// TIA Portal project "deneme1" (V16)

(* hardware
DEVICE "HMI_1"  TP1200 Comfort
   slot 0: "HMI_1"  TP1200 Comfort  6AV2 124-0MC01-0AX0  16.0.0.0
   slot 1: "HMI_RT_1"  TP1200 Comfort  6AV2 124-0MC01-0AX0  16.0.0.0
   slot 5: "HMI_1.IE_CP_1"  PROFINET Interface  16.0.0.0
      slot 1: "PROFINET Interface_1"  PROFINET Interface
         slot 1: "Port_1"  Port
         slot 2: "Port_2"  Port
   slot 7: "HMI_1.MPI/DP_CP_1"  MPI/DP Interface  16.0.0.0
DEVICE "S71500/ET200MP station_1"  S7-1500 station
   slot 0: "Rail_0"  Rack  6ES7 590-1***0-0AA0
   slot 1: "PLC_1"  CPU 1515-2 PN  6ES7 515-2AM00-0AB0  V1.8
      slot 3: "CPU display_1"  6ES7591-1BA00-0AA0
      slot 32768: "PROFINET interface_1"  X1
         slot 32769: "Port_1"  X1 P1
         slot 32770: "Port_2"  X1 P2
      slot 33024: "PROFINET interface_2"  X2
         slot 33025: "Port_1"  X2 P1
*)

// ===== PLC "PLC_1"  CPU 1515-2 PN =====

VAR_GLOBAL   // PLC tag table "Default tag table"
   "BulunduğuKat" AT %MW0 : Int;
   "Asansor0katta" AT %M2.0 : Bool;
   "Asansor1katta" AT %M2.1 : Bool;
   "Asansor3katta" AT %M2.2 : Bool;
   "Asansor2katta" AT %M2.3 : Bool;
   "P_TRIG1" AT %M2.4 : Bool;
   "AsansorAsagı" AT %M2.5 : Bool;
   "P_TRIG2" AT %M2.6 : Bool;
   "AsansorAcKat0" AT %M2.7 : Bool;
   "KapıAcık" AT %M3.0 : Bool;
   "P_TRIG3" AT %M3.1 : Bool;
   "AsansorKapatKat0" AT %M3.2 : Bool;
   "P_TRIG4" AT %M3.3 : Bool;
   "KapıKapalı" AT %M3.4 : Bool;
   "IsıkBariyeri" AT %M3.5 : Bool;
   "0KatDown" AT %M3.6 : Bool;
   "P_TRIG5" AT %M3.7 : Bool;
   "1KatGİT" AT %M4.0 : Bool;
   "2KatGİT" AT %M4.1 : Bool;
   "3KatGİT" AT %M4.2 : Bool;
   "AsansorYukarı" AT %M4.3 : Bool;
   "P_TRIG6" AT %M4.4 : Bool;
   "AsansorAcKat1" AT %M4.5 : Bool;
   "P_TRIG7" AT %M4.6 : Bool;
   "AsansorKapatKat1" AT %M4.7 : Bool;
   "P_TRIG8" AT %M5.0 : Bool;
   "P_TRIG9" AT %M5.1 : Bool;
   "P_TRIG10" AT %M5.2 : Bool;
   "AsansorAcKat2" AT %M5.3 : Bool;
   "P_TRIG11" AT %M5.4 : Bool;
   "P_TRIG12" AT %M5.5 : Bool;
   "AsansorAcKat3" AT %M5.6 : Bool;
   "1Katagit0dan" AT %M5.7 : Bool;
   "2katagit0dan" AT %M6.0 : Bool;
   "3katagit0dan" AT %M6.1 : Bool;
   "P_TRIG13" AT %M6.2 : Bool;
   "P_TRIG14" AT %M6.3 : Bool;
   "P_TRIG15" AT %M6.4 : Bool;
   "P_TRIG16" AT %M6.5 : Bool;
   "P_TRIG17" AT %M6.6 : Bool;
   "AsansorKapatKat2" AT %M6.7 : Bool;
   "AsansorKapatKat3" AT %M7.0 : Bool;
   "P_TRIG18" AT %M7.1 : Bool;
   "P_TRIG19" AT %M7.2 : Bool;
   "P_TRIG20" AT %M7.3 : Bool;
   "P_TRIG21" AT %M7.4 : Bool;
   "1KatDown" AT %M7.5 : Bool;
   "P_TRIG22" AT %M7.6 : Bool;
   "1KatUp" AT %M7.7 : Bool;
   "P_TRIG23" AT %M8.0 : Bool;
   "P_TRIG25" AT %M8.1 : Bool;
   "P_TRIG24" AT %M8.2 : Bool;
   "P_TRIG26" AT %M8.3 : Bool;
   "0KataGit" AT %M8.4 : Bool;
   "2katagit1den" AT %M8.5 : Bool;
   "3katagit1den" AT %M8.6 : Bool;
   "0katagit1den" AT %M8.7 : Bool;
   "P_TRIG27" AT %M9.0 : Bool;
   "P_TRIG28" AT %M9.1 : Bool;
   "P_TRIG29" AT %M9.2 : Bool;
   "P_TRIG30" AT %M9.3 : Bool;
   "P_TRIG31" AT %M9.4 : Bool;
   "P_TRIG32" AT %M9.5 : Bool;
   "P_TRIG33" AT %M9.6 : Bool;
   "P_TRIG34" AT %M9.7 : Bool;
   "P_TRIG35" AT %M10.0 : Bool;
   "P_TRIG36" AT %M10.1 : Bool;
   "P_TRIG37" AT %M10.2 : Bool;
   "P_TRIG38" AT %M10.3 : Bool;
   "P_TRIG39" AT %M10.4 : Bool;
   "P_TRIG40" AT %M10.5 : Bool;
   "Asansorsuan1katta" AT %M10.6 : Bool;
   "Asansorsuan0katta" AT %M10.7 : Bool;
   "P_TRIG41" AT %M11.0 : Bool;
   "P_TRIG42" AT %M11.1 : Bool;
   "P_TRIG43" AT %M11.2 : Bool;
   "P_TRIG44" AT %M11.3 : Bool;
   "P_TRIG45" AT %M11.4 : Bool;
   "P_TRIG46" AT %M11.5 : Bool;
   "P_TRIG47" AT %M11.6 : Bool;
   "P_TRIG48" AT %M11.7 : Bool;
   "P_TRIG49" AT %M12.0 : Bool;
   "P_TRIG50" AT %M12.1 : Bool;
   "P_TRIG51" AT %M12.2 : Bool;
   "P_TRIG52" AT %M12.3 : Bool;
   "P_TRIG53" AT %M12.4 : Bool;
   "P_TRIG54" AT %M12.5 : Bool;
   "P_TRIG55" AT %M12.6 : Bool;
   "P_TRIG56" AT %M12.7 : Bool;
   "deneme1" AT %M13.0 : Bool;
   "P_TRIG100" AT %M13.1 : Bool;
   "P_TRIG101" AT %M13.2 : Bool;
   "P_TRIG102" AT %M13.3 : Bool;
   "kapıacıkset" AT %M13.4 : Bool;
   "P_TRIG103" AT %M13.5 : Bool;
   "P_TRIG104" AT %M13.6 : Bool;
   "P_TRIG107" AT %M13.7 : Bool;
   "P_TRIG108" AT %M14.0 : Bool;
   "P_TRIG106" AT %M14.1 : Bool;
   "P_TRIG105" AT %M14.2 : Bool;
   "P_TRIG111" AT %M14.3 : Bool;
   "P_TRIG110" AT %M14.4 : Bool;
   "P_TRIG109" AT %M14.5 : Bool;
   "P_TRIG114" AT %M14.6 : Bool;
   "P_TRIG113" AT %M14.7 : Bool;
   "P_TRIG112" AT %M15.0 : Bool;
   "P_TRIG120" AT %M15.1 : Bool;
   "P_TRIG115" AT %M15.2 : Bool;
   "P_TRIG116" AT %M15.3 : Bool;
   "P_TRIG117" AT %M15.4 : Bool;
   "P_TRIG118" AT %M15.5 : Bool;
   "P_TRIG119" AT %M15.6 : Bool;
   "P_TRIG126" AT %M15.7 : Bool;
   "P_TRIG121" AT %M16.0 : Bool;
   "P_TRIG122" AT %M16.1 : Bool;
   "P_TRIG123" AT %M16.2 : Bool;
   "P_TRIG124" AT %M16.3 : Bool;
   "P_TRIG125" AT %M16.4 : Bool;
   "P_TRIG127" AT %M16.5 : Bool;
   "P_TRIG128" AT %M16.6 : Bool;
   "P_TRIG129" AT %M16.7 : Bool;
   "Asansorsuan2katta" AT %M17.0 : Bool;
   "P_TRIG130" AT %M17.6 : Bool;
   "P_TRIG131" AT %M17.1 : Bool;
   "P_TRIG132" AT %M17.2 : Bool;
   "P_TRIG133" AT %M17.5 : Bool;
   "P_TRIG134" AT %M17.3 : Bool;
   "P_TRIG135" AT %M17.4 : Bool;
   "3katagit2den" AT %M17.7 : Bool;
   "1katagit2den" AT %M18.0 : Bool;
   "0katagit2den" AT %M18.1 : Bool;
   "P_TRIG138" AT %M18.6 : Bool;
   "P_TRIG136" AT %M18.2 : Bool;
   "P_TRIG137" AT %M18.7 : Bool;
   "P_TRIG139" AT %M19.0 : Bool;
   "P_TRIG140" AT %M18.3 : Bool;
   "P_TRIG141" AT %M18.4 : Bool;
   "P_TRIG142" AT %M18.5 : Bool;
   "P_TRIG144" AT %M19.1 : Bool;
   "P_TRIG143" AT %M19.2 : Bool;
   "P_TRIG145" AT %M19.3 : Bool;
   "P_TRIG146" AT %M19.4 : Bool;
   "P_TRIG147" AT %M19.5 : Bool;
   "P_TRIG148" AT %M19.6 : Bool;
   "P_TRIG149" AT %M20.3 : Bool;
   "P_TRIG150" AT %M19.7 : Bool;
   "P_TRIG151" AT %M20.0 : Bool;
   "P_TRIG152" AT %M20.1 : Bool;
   "P_TRIG153" AT %M20.2 : Bool;
   "P_TRIG154" AT %M20.4 : Bool;
   "P_TRIG155" AT %M20.5 : Bool;
   "P_TRIG156" AT %M20.6 : Bool;
   "3katUp" AT %M20.7 : Bool;
   "Asansorsuan3katta" AT %M21.0 : Bool;
   "2katagit3den" AT %M21.1 : Bool;
   "1katagit3den" AT %M21.2 : Bool;
   "0katagit3den" AT %M21.3 : Bool;
   "P_TRIG164" AT %M21.4 : Bool;
   "P_TRIG163" AT %M22.0 : Bool;
   "P_TRIG162" AT %M21.5 : Bool;
   "P_TRIG161" AT %M21.6 : Bool;
   "P_TRIG160" AT %M21.7 : Bool;
   "P_TRIG171" AT %M22.1 : Bool;
   "P_TRIG170" AT %M22.2 : Bool;
   "P_TRIG169" AT %M22.7 : Bool;
   "P_TRIG168" AT %M22.3 : Bool;
   "P_TRIG167" AT %M22.4 : Bool;
   "P_TRIG166" AT %M22.5 : Bool;
   "P_TRIG165" AT %M22.6 : Bool;
   "P_TRIG172" AT %M23.0 : Bool;
   "P_TRIG173" AT %M23.1 : Bool;
   "P_TRIG174" AT %M23.2 : Bool;
   "P_TRIG175" AT %M23.3 : Bool;
   "P_TRIG176" AT %M23.4 : Bool;
   "P_TRIG177" AT %M23.5 : Bool;
   "P_TRIG178" AT %M23.6 : Bool;
   "P_TRIG179" AT %M23.7 : Bool;
   "P_TRIG180" AT %M24.0 : Bool;
   "P_TRIG181" AT %M24.1 : Bool;
   "P_TRIG182" AT %M24.2 : Bool;
   "P_TRIG183" AT %M24.3 : Bool;
   "P_TRIG184" AT %M24.4 : Bool;
   "P_TRIG185" AT %M24.5 : Bool;
   "P_TRIG186" AT %M24.6 : Bool;
   "2KatDown" AT %M24.7 : Bool;
   "2KatUp" AT %M25.0 : Bool;
END_VAR

ORGANIZATION_BLOCK "Main"   // OB1, LAD, ProgramCycle
TITLE = "Main Program Sweep (Cycle)"
{ S7_Optimized_Access := 'TRUE' }
VERSION : 0.1
   VAR_INPUT
      Initial_Call : Bool;   // Initial call of this OB
      Remanence : Bool;   // =True, if remanent data are available
   END_VAR
   VAR_TEMP   // added for the SCL form of the ladder/FBD networks
      _w1 : Bool;
      _w2 : Bool;
      _w3 : Bool;
      _w4 : Bool;
      _w5 : Bool;
      _w6 : Bool;
      _w7 : Bool;
      _w8 : Bool;
      _w9 : Bool;
      _w10 : Bool;
      _w11 : Bool;
      _w12 : Bool;
      _w13 : Bool;
      _w14 : Bool;
      _w15 : Bool;
      _w16 : Bool;
      _w17 : Bool;
      _w18 : Bool;
      _w19 : Bool;
      _w20 : Bool;
      _w21 : Bool;
      _w22 : Bool;
      _w23 : Bool;
      _w24 : Bool;
      _w25 : Bool;
      _w26 : Bool;
      _w27 : Bool;
      _w28 : Bool;
      _w29 : Bool;
      _w30 : Bool;
      _w31 : Bool;
      _w32 : Bool;
      _w33 : Bool;
      _w34 : Bool;
      _w35 : Bool;
      _w36 : Bool;
      _w37 : Bool;
      _w38 : Bool;
      _w39 : Bool;
      _w40 : Bool;
      _w41 : Bool;
      _w42 : Bool;
      _w43 : Bool;
      _w44 : Bool;
      _w45 : Bool;
      _w46 : Bool;
      _w47 : Bool;
      _w48 : Bool;
      _w49 : Bool;
      _w50 : Bool;
      _w51 : Bool;
      _w52 : Bool;
      _w53 : Bool;
      _w54 : Bool;
      _w55 : Bool;
   END_VAR
BEGIN

REGION Network 1: 0 a bas 1 2 3 den asansör gelsin
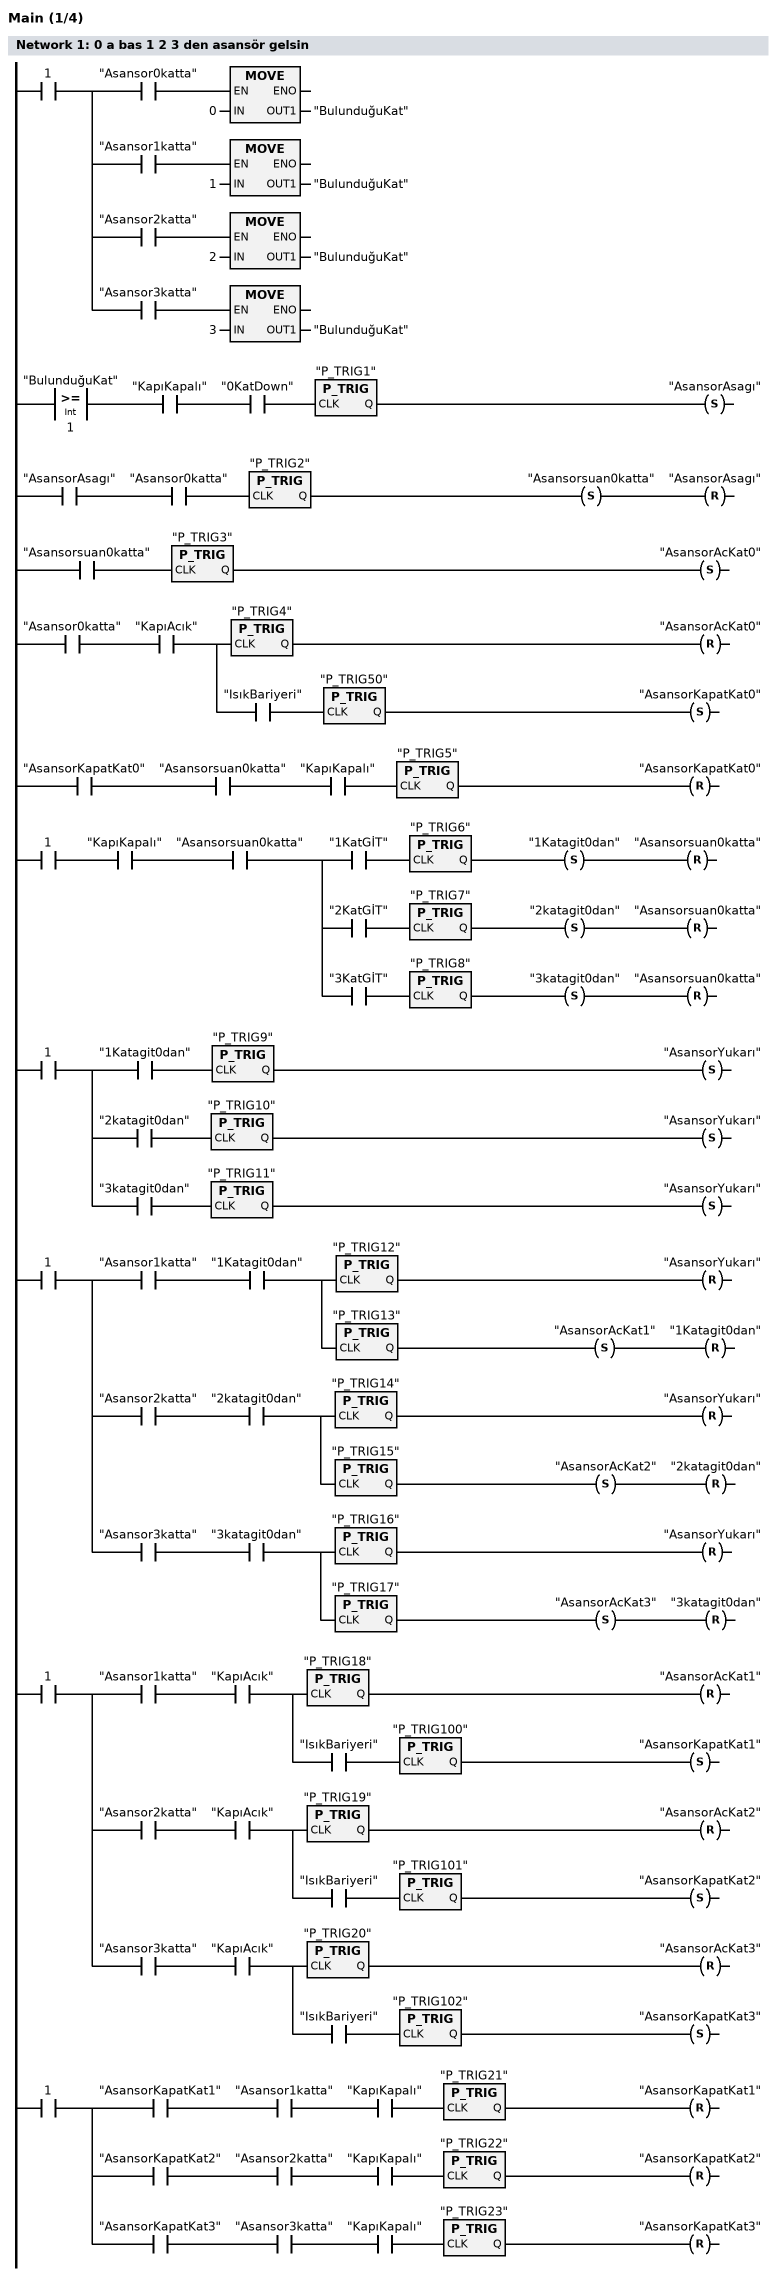
   RUNG wire#powerrail
      Contact( 1 )
      wire#w1
      Contact( "Asansor0katta" )
      Move(in := 0, out1 => "BulunduğuKat")
   END_RUNG
   RUNG wire#w1
      Contact( "Asansor1katta" )
      Move(in := 1, out1 => "BulunduğuKat")
   END_RUNG
   RUNG wire#w1
      Contact( "Asansor2katta" )
      Move(in := 2, out1 => "BulunduğuKat")
   END_RUNG
   RUNG wire#w1
      Contact( "Asansor3katta" )
      Move(in := 3, out1 => "BulunduğuKat")
   END_RUNG
   RUNG wire#powerrail
      { S7_Templates := "SrcType := Int" } GE_Contact(in1 := "BulunduğuKat", in2 := 1)
      Contact( "KapıKapalı" )
      Contact( "0KatDown" )
      P_Trig( "P_TRIG1" )
      S_Coil( "AsansorAsagı" )
   END_RUNG
   RUNG wire#powerrail
      Contact( "AsansorAsagı" )
      Contact( "Asansor0katta" )
      P_Trig( "P_TRIG2" )
      S_Coil( "Asansorsuan0katta" )
      R_Coil( "AsansorAsagı" )
   END_RUNG
   RUNG wire#powerrail
      Contact( "Asansorsuan0katta" )
      P_Trig( "P_TRIG3" )
      S_Coil( "AsansorAcKat0" )
   END_RUNG
   RUNG wire#powerrail
      Contact( "Asansor0katta" )
      Contact( "KapıAcık" )
      wire#w2
      P_Trig( "P_TRIG4" )
      R_Coil( "AsansorAcKat0" )
   END_RUNG
   RUNG wire#w2
      Contact( "IsıkBariyeri" )
      P_Trig( "P_TRIG50" )
      S_Coil( "AsansorKapatKat0" )
   END_RUNG
   RUNG wire#powerrail
      Contact( "AsansorKapatKat0" )
      Contact( "Asansorsuan0katta" )
      Contact( "KapıKapalı" )
      P_Trig( "P_TRIG5" )
      R_Coil( "AsansorKapatKat0" )
   END_RUNG
   RUNG wire#powerrail
      Contact( 1 )
      Contact( "KapıKapalı" )
      Contact( "Asansorsuan0katta" )
      wire#w3
      Contact( "1KatGİT" )
      P_Trig( "P_TRIG6" )
      S_Coil( "1Katagit0dan" )
      R_Coil( "Asansorsuan0katta" )
   END_RUNG
   RUNG wire#w3
      Contact( "2KatGİT" )
      P_Trig( "P_TRIG7" )
      S_Coil( "2katagit0dan" )
      R_Coil( "Asansorsuan0katta" )
   END_RUNG
   RUNG wire#w3
      Contact( "3KatGİT" )
      P_Trig( "P_TRIG8" )
      S_Coil( "3katagit0dan" )
      R_Coil( "Asansorsuan0katta" )
   END_RUNG
   RUNG wire#powerrail
      Contact( 1 )
      wire#w4
      Contact( "1Katagit0dan" )
      P_Trig( "P_TRIG9" )
      S_Coil( "AsansorYukarı" )
   END_RUNG
   RUNG wire#w4
      Contact( "2katagit0dan" )
      P_Trig( "P_TRIG10" )
      S_Coil( "AsansorYukarı" )
   END_RUNG
   RUNG wire#w4
      Contact( "3katagit0dan" )
      P_Trig( "P_TRIG11" )
      S_Coil( "AsansorYukarı" )
   END_RUNG
   RUNG wire#powerrail
      Contact( 1 )
      wire#w5
      Contact( "Asansor1katta" )
      Contact( "1Katagit0dan" )
      wire#w6
      P_Trig( "P_TRIG12" )
      R_Coil( "AsansorYukarı" )
   END_RUNG
   RUNG wire#w6
      P_Trig( "P_TRIG13" )
      S_Coil( "AsansorAcKat1" )
      R_Coil( "1Katagit0dan" )
   END_RUNG
   RUNG wire#w5
      Contact( "Asansor2katta" )
      Contact( "2katagit0dan" )
      wire#w7
      P_Trig( "P_TRIG14" )
      R_Coil( "AsansorYukarı" )
   END_RUNG
   RUNG wire#w7
      P_Trig( "P_TRIG15" )
      S_Coil( "AsansorAcKat2" )
      R_Coil( "2katagit0dan" )
   END_RUNG
   RUNG wire#w5
      Contact( "Asansor3katta" )
      Contact( "3katagit0dan" )
      wire#w8
      P_Trig( "P_TRIG16" )
      R_Coil( "AsansorYukarı" )
   END_RUNG
   RUNG wire#w8
      P_Trig( "P_TRIG17" )
      S_Coil( "AsansorAcKat3" )
      R_Coil( "3katagit0dan" )
   END_RUNG
   RUNG wire#powerrail
      Contact( 1 )
      wire#w9
      Contact( "Asansor1katta" )
      Contact( "KapıAcık" )
      wire#w10
      P_Trig( "P_TRIG18" )
      R_Coil( "AsansorAcKat1" )
   END_RUNG
   RUNG wire#w10
      Contact( "IsıkBariyeri" )
      P_Trig( "P_TRIG100" )
      S_Coil( "AsansorKapatKat1" )
   END_RUNG
   RUNG wire#w9
      Contact( "Asansor2katta" )
      Contact( "KapıAcık" )
      wire#w11
      P_Trig( "P_TRIG19" )
      R_Coil( "AsansorAcKat2" )
   END_RUNG
   RUNG wire#w11
      Contact( "IsıkBariyeri" )
      P_Trig( "P_TRIG101" )
      S_Coil( "AsansorKapatKat2" )
   END_RUNG
   RUNG wire#w9
      Contact( "Asansor3katta" )
      Contact( "KapıAcık" )
      wire#w12
      P_Trig( "P_TRIG20" )
      R_Coil( "AsansorAcKat3" )
   END_RUNG
   RUNG wire#w12
      Contact( "IsıkBariyeri" )
      P_Trig( "P_TRIG102" )
      S_Coil( "AsansorKapatKat3" )
   END_RUNG
   RUNG wire#powerrail
      Contact( 1 )
      wire#w13
      Contact( "AsansorKapatKat1" )
      Contact( "Asansor1katta" )
      Contact( "KapıKapalı" )
      P_Trig( "P_TRIG21" )
      R_Coil( "AsansorKapatKat1" )
   END_RUNG
   RUNG wire#w13
      Contact( "AsansorKapatKat2" )
      Contact( "Asansor2katta" )
      Contact( "KapıKapalı" )
      P_Trig( "P_TRIG22" )
      R_Coil( "AsansorKapatKat2" )
   END_RUNG
   RUNG wire#w13
      Contact( "AsansorKapatKat3" )
      Contact( "Asansor3katta" )
      Contact( "KapıKapalı" )
      P_Trig( "P_TRIG23" )
      R_Coil( "AsansorKapatKat3" )
   END_RUNG
   // the same network as SCL:
   IF 1 AND "Asansor0katta" THEN "BulunduğuKat" := 0; END_IF;
   IF 1 AND "Asansor1katta" THEN "BulunduğuKat" := 1; END_IF;
   IF 1 AND "Asansor2katta" THEN "BulunduğuKat" := 2; END_IF;
   IF 1 AND "Asansor3katta" THEN "BulunduğuKat" := 3; END_IF;
   #_w1 := ("BulunduğuKat" >= 1) AND "KapıKapalı" AND "0KatDown";
   #_w2 := #_w1 AND NOT "P_TRIG1";   // rising edge
   "P_TRIG1" := #_w1;
   IF #_w2 THEN "AsansorAsagı" := TRUE; END_IF;
   #_w3 := "AsansorAsagı" AND "Asansor0katta";
   #_w4 := #_w3 AND NOT "P_TRIG2";   // rising edge
   "P_TRIG2" := #_w3;
   IF #_w4 THEN
       "Asansorsuan0katta" := TRUE;
       "AsansorAsagı" := FALSE;
   END_IF;
   #_w5 := "Asansorsuan0katta" AND NOT "P_TRIG3";   // rising edge
   "P_TRIG3" := "Asansorsuan0katta";
   IF #_w5 THEN "AsansorAcKat0" := TRUE; END_IF;
   #_w6 := "Asansor0katta" AND "KapıAcık";
   #_w7 := #_w6 AND NOT "P_TRIG4";   // rising edge
   "P_TRIG4" := #_w6;
   IF #_w7 THEN "AsansorAcKat0" := FALSE; END_IF;
   #_w8 := #_w6 AND "IsıkBariyeri";
   #_w9 := #_w8 AND NOT "P_TRIG50";   // rising edge
   "P_TRIG50" := #_w8;
   IF #_w9 THEN "AsansorKapatKat0" := TRUE; END_IF;
   #_w10 := "AsansorKapatKat0" AND "Asansorsuan0katta" AND "KapıKapalı";
   #_w11 := #_w10 AND NOT "P_TRIG5";   // rising edge
   "P_TRIG5" := #_w10;
   IF #_w11 THEN "AsansorKapatKat0" := FALSE; END_IF;
   #_w12 := 1 AND "KapıKapalı" AND "Asansorsuan0katta";
   #_w13 := #_w12 AND "1KatGİT";
   #_w14 := #_w13 AND NOT "P_TRIG6";   // rising edge
   "P_TRIG6" := #_w13;
   IF #_w14 THEN
       "1Katagit0dan" := TRUE;
       "Asansorsuan0katta" := FALSE;
   END_IF;
   #_w15 := #_w12 AND "2KatGİT";
   #_w16 := #_w15 AND NOT "P_TRIG7";   // rising edge
   "P_TRIG7" := #_w15;
   IF #_w16 THEN
       "2katagit0dan" := TRUE;
       "Asansorsuan0katta" := FALSE;
   END_IF;
   #_w17 := #_w12 AND "3KatGİT";
   #_w18 := #_w17 AND NOT "P_TRIG8";   // rising edge
   "P_TRIG8" := #_w17;
   IF #_w18 THEN
       "3katagit0dan" := TRUE;
       "Asansorsuan0katta" := FALSE;
   END_IF;
   #_w19 := 1 AND "1Katagit0dan";
   #_w20 := #_w19 AND NOT "P_TRIG9";   // rising edge
   "P_TRIG9" := #_w19;
   IF #_w20 THEN "AsansorYukarı" := TRUE; END_IF;
   #_w21 := 1 AND "2katagit0dan";
   #_w22 := #_w21 AND NOT "P_TRIG10";   // rising edge
   "P_TRIG10" := #_w21;
   IF #_w22 THEN "AsansorYukarı" := TRUE; END_IF;
   #_w23 := 1 AND "3katagit0dan";
   #_w24 := #_w23 AND NOT "P_TRIG11";   // rising edge
   "P_TRIG11" := #_w23;
   IF #_w24 THEN "AsansorYukarı" := TRUE; END_IF;
   #_w25 := 1 AND "Asansor1katta" AND "1Katagit0dan";
   #_w26 := #_w25 AND NOT "P_TRIG12";   // rising edge
   "P_TRIG12" := #_w25;
   IF #_w26 THEN "AsansorYukarı" := FALSE; END_IF;
   #_w27 := #_w25 AND NOT "P_TRIG13";   // rising edge
   "P_TRIG13" := #_w25;
   IF #_w27 THEN
       "AsansorAcKat1" := TRUE;
       "1Katagit0dan" := FALSE;
   END_IF;
   #_w28 := 1 AND "Asansor2katta" AND "2katagit0dan";
   #_w29 := #_w28 AND NOT "P_TRIG14";   // rising edge
   "P_TRIG14" := #_w28;
   IF #_w29 THEN "AsansorYukarı" := FALSE; END_IF;
   #_w30 := #_w28 AND NOT "P_TRIG15";   // rising edge
   "P_TRIG15" := #_w28;
   IF #_w30 THEN
       "AsansorAcKat2" := TRUE;
       "2katagit0dan" := FALSE;
   END_IF;
   #_w31 := 1 AND "Asansor3katta" AND "3katagit0dan";
   #_w32 := #_w31 AND NOT "P_TRIG16";   // rising edge
   "P_TRIG16" := #_w31;
   IF #_w32 THEN "AsansorYukarı" := FALSE; END_IF;
   #_w33 := #_w31 AND NOT "P_TRIG17";   // rising edge
   "P_TRIG17" := #_w31;
   IF #_w33 THEN
       "AsansorAcKat3" := TRUE;
       "3katagit0dan" := FALSE;
   END_IF;
   #_w34 := 1 AND "Asansor1katta" AND "KapıAcık";
   #_w35 := #_w34 AND NOT "P_TRIG18";   // rising edge
   "P_TRIG18" := #_w34;
   IF #_w35 THEN "AsansorAcKat1" := FALSE; END_IF;
   #_w36 := #_w34 AND "IsıkBariyeri";
   #_w37 := #_w36 AND NOT "P_TRIG100";   // rising edge
   "P_TRIG100" := #_w36;
   IF #_w37 THEN "AsansorKapatKat1" := TRUE; END_IF;
   #_w38 := 1 AND "Asansor2katta" AND "KapıAcık";
   #_w39 := #_w38 AND NOT "P_TRIG19";   // rising edge
   "P_TRIG19" := #_w38;
   IF #_w39 THEN "AsansorAcKat2" := FALSE; END_IF;
   #_w40 := #_w38 AND "IsıkBariyeri";
   #_w41 := #_w40 AND NOT "P_TRIG101";   // rising edge
   "P_TRIG101" := #_w40;
   IF #_w41 THEN "AsansorKapatKat2" := TRUE; END_IF;
   #_w42 := 1 AND "Asansor3katta" AND "KapıAcık";
   #_w43 := #_w42 AND NOT "P_TRIG20";   // rising edge
   "P_TRIG20" := #_w42;
   IF #_w43 THEN "AsansorAcKat3" := FALSE; END_IF;
   #_w44 := #_w42 AND "IsıkBariyeri";
   #_w45 := #_w44 AND NOT "P_TRIG102";   // rising edge
   "P_TRIG102" := #_w44;
   IF #_w45 THEN "AsansorKapatKat3" := TRUE; END_IF;
   #_w46 := 1 AND "AsansorKapatKat1" AND "Asansor1katta" AND "KapıKapalı";
   #_w47 := #_w46 AND NOT "P_TRIG21";   // rising edge
   "P_TRIG21" := #_w46;
   IF #_w47 THEN "AsansorKapatKat1" := FALSE; END_IF;
   #_w48 := 1 AND "AsansorKapatKat2" AND "Asansor2katta" AND "KapıKapalı";
   #_w49 := #_w48 AND NOT "P_TRIG22";   // rising edge
   "P_TRIG22" := #_w48;
   IF #_w49 THEN "AsansorKapatKat2" := FALSE; END_IF;
   #_w50 := 1 AND "AsansorKapatKat3" AND "Asansor3katta" AND "KapıKapalı";
   #_w51 := #_w50 AND NOT "P_TRIG23";   // rising edge
   "P_TRIG23" := #_w50;
   IF #_w51 THEN "AsansorKapatKat3" := FALSE; END_IF;
END_REGION

REGION Network 2: 1 katda iken 0 dan çağırma veya 1 katda iken 2 ve 3 den cağırma
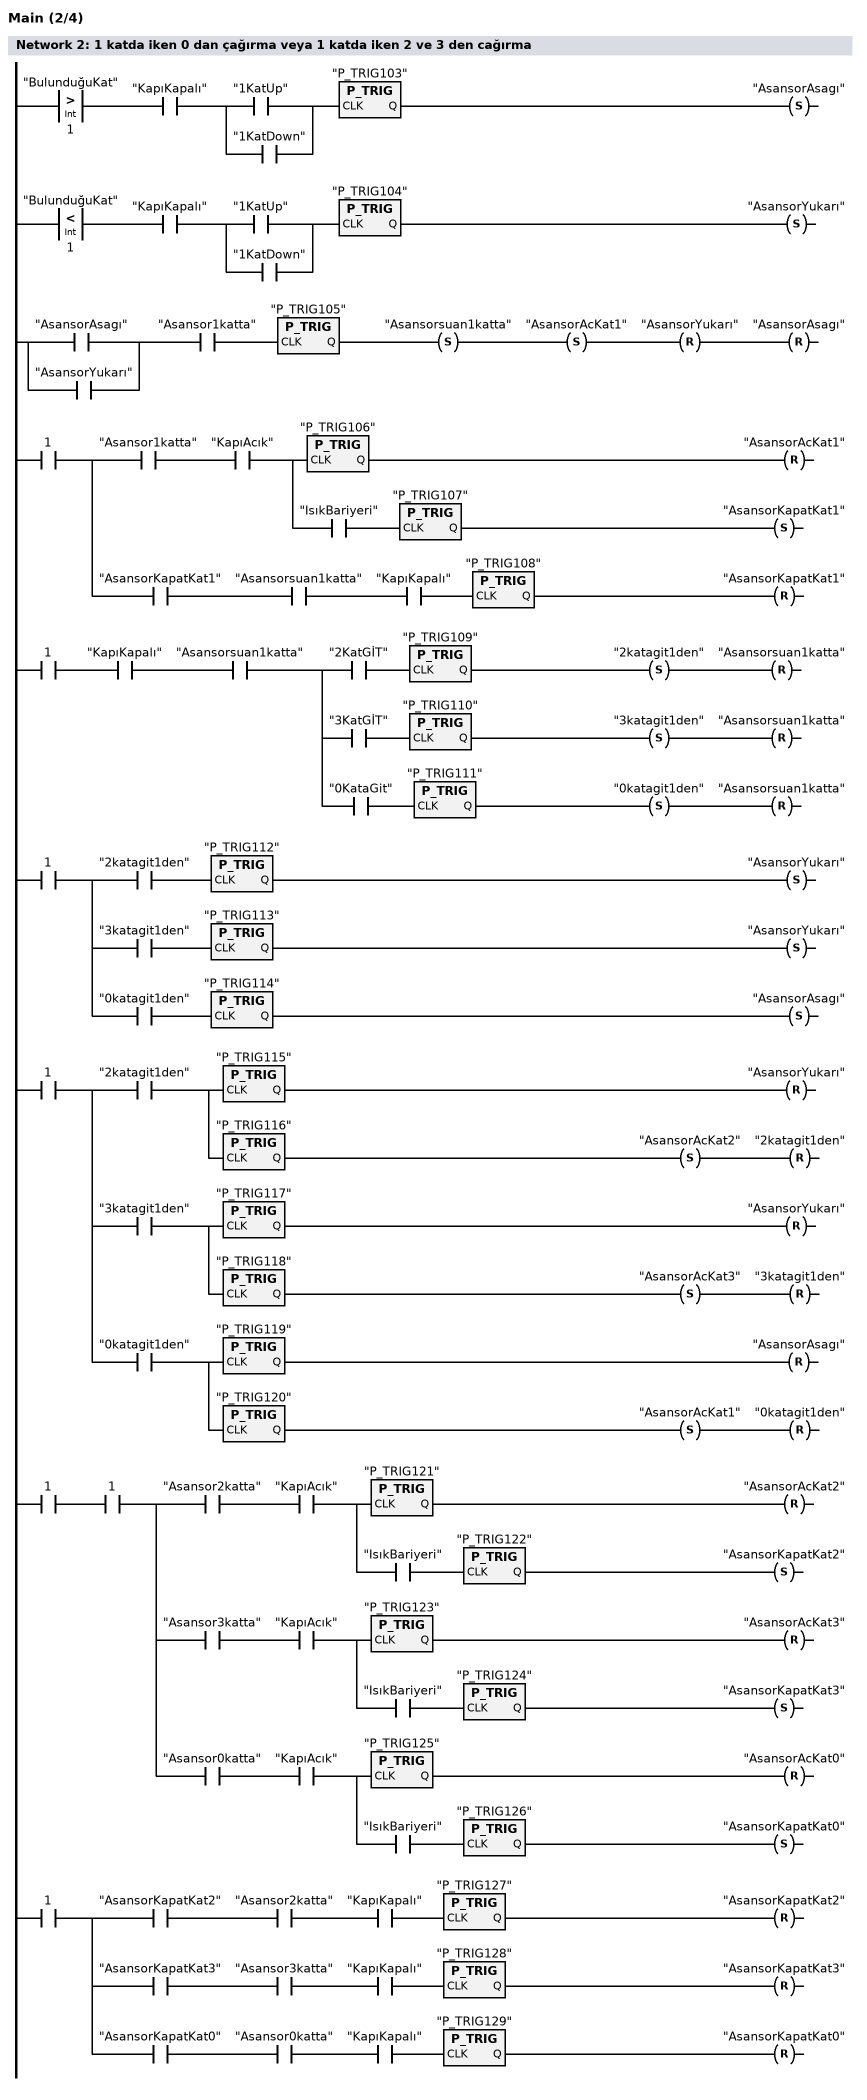
   RUNG wire#powerrail
      { S7_Templates := "SrcType := Int" } GT_Contact(in1 := "BulunduğuKat", in2 := 1)
      Contact( "KapıKapalı" )
      wire#w1
      Contact( "1KatUp" )
      wire#w2
      P_Trig( "P_TRIG103" )
      S_Coil( "AsansorAsagı" )
   END_RUNG
   RUNG wire#w1
      Contact( "1KatDown" )
   END_RUNG wire#w2
   RUNG wire#powerrail
      { S7_Templates := "SrcType := Int" } LT_Contact(in1 := "BulunduğuKat", in2 := 1)
      Contact( "KapıKapalı" )
      wire#w3
      Contact( "1KatUp" )
      wire#w4
      P_Trig( "P_TRIG104" )
      S_Coil( "AsansorYukarı" )
   END_RUNG
   RUNG wire#w3
      Contact( "1KatDown" )
   END_RUNG wire#w4
   RUNG wire#powerrail
      Contact( "AsansorAsagı" )
      wire#w5
      Contact( "Asansor1katta" )
      P_Trig( "P_TRIG105" )
      S_Coil( "Asansorsuan1katta" )
      S_Coil( "AsansorAcKat1" )
      R_Coil( "AsansorYukarı" )
      R_Coil( "AsansorAsagı" )
   END_RUNG
   RUNG wire#powerrail
      Contact( "AsansorYukarı" )
   END_RUNG wire#w5
   RUNG wire#powerrail
      Contact( 1 )
      wire#w6
      Contact( "Asansor1katta" )
      Contact( "KapıAcık" )
      wire#w7
      P_Trig( "P_TRIG106" )
      R_Coil( "AsansorAcKat1" )
   END_RUNG
   RUNG wire#w7
      Contact( "IsıkBariyeri" )
      P_Trig( "P_TRIG107" )
      S_Coil( "AsansorKapatKat1" )
   END_RUNG
   RUNG wire#w6
      Contact( "AsansorKapatKat1" )
      Contact( "Asansorsuan1katta" )
      Contact( "KapıKapalı" )
      P_Trig( "P_TRIG108" )
      R_Coil( "AsansorKapatKat1" )
   END_RUNG
   RUNG wire#powerrail
      Contact( 1 )
      Contact( "KapıKapalı" )
      Contact( "Asansorsuan1katta" )
      wire#w8
      Contact( "2KatGİT" )
      P_Trig( "P_TRIG109" )
      S_Coil( "2katagit1den" )
      R_Coil( "Asansorsuan1katta" )
   END_RUNG
   RUNG wire#w8
      Contact( "3KatGİT" )
      P_Trig( "P_TRIG110" )
      S_Coil( "3katagit1den" )
      R_Coil( "Asansorsuan1katta" )
   END_RUNG
   RUNG wire#w8
      Contact( "0KataGit" )
      P_Trig( "P_TRIG111" )
      S_Coil( "0katagit1den" )
      R_Coil( "Asansorsuan1katta" )
   END_RUNG
   RUNG wire#powerrail
      Contact( 1 )
      wire#w9
      Contact( "2katagit1den" )
      P_Trig( "P_TRIG112" )
      S_Coil( "AsansorYukarı" )
   END_RUNG
   RUNG wire#w9
      Contact( "3katagit1den" )
      P_Trig( "P_TRIG113" )
      S_Coil( "AsansorYukarı" )
   END_RUNG
   RUNG wire#w9
      Contact( "0katagit1den" )
      P_Trig( "P_TRIG114" )
      S_Coil( "AsansorAsagı" )
   END_RUNG
   RUNG wire#powerrail
      Contact( 1 )
      wire#w10
      Contact( "2katagit1den" )
      wire#w11
      P_Trig( "P_TRIG115" )
      R_Coil( "AsansorYukarı" )
   END_RUNG
   RUNG wire#w11
      P_Trig( "P_TRIG116" )
      S_Coil( "AsansorAcKat2" )
      R_Coil( "2katagit1den" )
   END_RUNG
   RUNG wire#w10
      Contact( "3katagit1den" )
      wire#w12
      P_Trig( "P_TRIG117" )
      R_Coil( "AsansorYukarı" )
   END_RUNG
   RUNG wire#w12
      P_Trig( "P_TRIG118" )
      S_Coil( "AsansorAcKat3" )
      R_Coil( "3katagit1den" )
   END_RUNG
   RUNG wire#w10
      Contact( "0katagit1den" )
      wire#w13
      P_Trig( "P_TRIG119" )
      R_Coil( "AsansorAsagı" )
   END_RUNG
   RUNG wire#w13
      P_Trig( "P_TRIG120" )
      S_Coil( "AsansorAcKat1" )
      R_Coil( "0katagit1den" )
   END_RUNG
   RUNG wire#powerrail
      Contact( 1 )
      Contact( 1 )
      wire#w14
      Contact( "Asansor2katta" )
      Contact( "KapıAcık" )
      wire#w15
      P_Trig( "P_TRIG121" )
      R_Coil( "AsansorAcKat2" )
   END_RUNG
   RUNG wire#w15
      Contact( "IsıkBariyeri" )
      P_Trig( "P_TRIG122" )
      S_Coil( "AsansorKapatKat2" )
   END_RUNG
   RUNG wire#w14
      Contact( "Asansor3katta" )
      Contact( "KapıAcık" )
      wire#w16
      P_Trig( "P_TRIG123" )
      R_Coil( "AsansorAcKat3" )
   END_RUNG
   RUNG wire#w16
      Contact( "IsıkBariyeri" )
      P_Trig( "P_TRIG124" )
      S_Coil( "AsansorKapatKat3" )
   END_RUNG
   RUNG wire#w14
      Contact( "Asansor0katta" )
      Contact( "KapıAcık" )
      wire#w17
      P_Trig( "P_TRIG125" )
      R_Coil( "AsansorAcKat0" )
   END_RUNG
   RUNG wire#w17
      Contact( "IsıkBariyeri" )
      P_Trig( "P_TRIG126" )
      S_Coil( "AsansorKapatKat0" )
   END_RUNG
   RUNG wire#powerrail
      Contact( 1 )
      wire#w18
      Contact( "AsansorKapatKat2" )
      Contact( "Asansor2katta" )
      Contact( "KapıKapalı" )
      P_Trig( "P_TRIG127" )
      R_Coil( "AsansorKapatKat2" )
   END_RUNG
   RUNG wire#w18
      Contact( "AsansorKapatKat3" )
      Contact( "Asansor3katta" )
      Contact( "KapıKapalı" )
      P_Trig( "P_TRIG128" )
      R_Coil( "AsansorKapatKat3" )
   END_RUNG
   RUNG wire#w18
      Contact( "AsansorKapatKat0" )
      Contact( "Asansor0katta" )
      Contact( "KapıKapalı" )
      P_Trig( "P_TRIG129" )
      R_Coil( "AsansorKapatKat0" )
   END_RUNG
   // the same network as SCL:
   #_w1 := ("BulunduğuKat" > 1) AND "KapıKapalı" AND ("1KatUp" OR "1KatDown");
   #_w2 := #_w1 AND NOT "P_TRIG103";   // rising edge
   "P_TRIG103" := #_w1;
   IF #_w2 THEN "AsansorAsagı" := TRUE; END_IF;
   #_w3 := ("BulunduğuKat" < 1) AND "KapıKapalı" AND ("1KatUp" OR "1KatDown");
   #_w4 := #_w3 AND NOT "P_TRIG104";   // rising edge
   "P_TRIG104" := #_w3;
   IF #_w4 THEN "AsansorYukarı" := TRUE; END_IF;
   #_w5 := ("AsansorAsagı" OR "AsansorYukarı") AND "Asansor1katta";
   #_w6 := #_w5 AND NOT "P_TRIG105";   // rising edge
   "P_TRIG105" := #_w5;
   IF #_w6 THEN
       "Asansorsuan1katta" := TRUE;
       "AsansorAcKat1" := TRUE;
       "AsansorYukarı" := FALSE;
       "AsansorAsagı" := FALSE;
   END_IF;
   #_w7 := 1 AND "Asansor1katta" AND "KapıAcık";
   #_w8 := #_w7 AND NOT "P_TRIG106";   // rising edge
   "P_TRIG106" := #_w7;
   IF #_w8 THEN "AsansorAcKat1" := FALSE; END_IF;
   #_w9 := #_w7 AND "IsıkBariyeri";
   #_w10 := #_w9 AND NOT "P_TRIG107";   // rising edge
   "P_TRIG107" := #_w9;
   IF #_w10 THEN "AsansorKapatKat1" := TRUE; END_IF;
   #_w11 := 1 AND "AsansorKapatKat1" AND "Asansorsuan1katta" AND "KapıKapalı";
   #_w12 := #_w11 AND NOT "P_TRIG108";   // rising edge
   "P_TRIG108" := #_w11;
   IF #_w12 THEN "AsansorKapatKat1" := FALSE; END_IF;
   #_w13 := 1 AND "KapıKapalı" AND "Asansorsuan1katta";
   #_w14 := #_w13 AND "2KatGİT";
   #_w15 := #_w14 AND NOT "P_TRIG109";   // rising edge
   "P_TRIG109" := #_w14;
   IF #_w15 THEN
       "2katagit1den" := TRUE;
       "Asansorsuan1katta" := FALSE;
   END_IF;
   #_w16 := #_w13 AND "3KatGİT";
   #_w17 := #_w16 AND NOT "P_TRIG110";   // rising edge
   "P_TRIG110" := #_w16;
   IF #_w17 THEN
       "3katagit1den" := TRUE;
       "Asansorsuan1katta" := FALSE;
   END_IF;
   #_w18 := #_w13 AND "0KataGit";
   #_w19 := #_w18 AND NOT "P_TRIG111";   // rising edge
   "P_TRIG111" := #_w18;
   IF #_w19 THEN
       "0katagit1den" := TRUE;
       "Asansorsuan1katta" := FALSE;
   END_IF;
   #_w20 := 1 AND "2katagit1den";
   #_w21 := #_w20 AND NOT "P_TRIG112";   // rising edge
   "P_TRIG112" := #_w20;
   IF #_w21 THEN "AsansorYukarı" := TRUE; END_IF;
   #_w22 := 1 AND "3katagit1den";
   #_w23 := #_w22 AND NOT "P_TRIG113";   // rising edge
   "P_TRIG113" := #_w22;
   IF #_w23 THEN "AsansorYukarı" := TRUE; END_IF;
   #_w24 := 1 AND "0katagit1den";
   #_w25 := #_w24 AND NOT "P_TRIG114";   // rising edge
   "P_TRIG114" := #_w24;
   IF #_w25 THEN "AsansorAsagı" := TRUE; END_IF;
   #_w26 := 1 AND "2katagit1den";
   #_w27 := #_w26 AND NOT "P_TRIG115";   // rising edge
   "P_TRIG115" := #_w26;
   IF #_w27 THEN "AsansorYukarı" := FALSE; END_IF;
   #_w28 := #_w26 AND NOT "P_TRIG116";   // rising edge
   "P_TRIG116" := #_w26;
   IF #_w28 THEN
       "AsansorAcKat2" := TRUE;
       "2katagit1den" := FALSE;
   END_IF;
   #_w29 := 1 AND "3katagit1den";
   #_w30 := #_w29 AND NOT "P_TRIG117";   // rising edge
   "P_TRIG117" := #_w29;
   IF #_w30 THEN "AsansorYukarı" := FALSE; END_IF;
   #_w31 := #_w29 AND NOT "P_TRIG118";   // rising edge
   "P_TRIG118" := #_w29;
   IF #_w31 THEN
       "AsansorAcKat3" := TRUE;
       "3katagit1den" := FALSE;
   END_IF;
   #_w32 := 1 AND "0katagit1den";
   #_w33 := #_w32 AND NOT "P_TRIG119";   // rising edge
   "P_TRIG119" := #_w32;
   IF #_w33 THEN "AsansorAsagı" := FALSE; END_IF;
   #_w34 := #_w32 AND NOT "P_TRIG120";   // rising edge
   "P_TRIG120" := #_w32;
   IF #_w34 THEN
       "AsansorAcKat1" := TRUE;
       "0katagit1den" := FALSE;
   END_IF;
   #_w35 := 1 AND 1;
   #_w36 := #_w35 AND "Asansor2katta" AND "KapıAcık";
   #_w37 := #_w36 AND NOT "P_TRIG121";   // rising edge
   "P_TRIG121" := #_w36;
   IF #_w37 THEN "AsansorAcKat2" := FALSE; END_IF;
   #_w38 := #_w36 AND "IsıkBariyeri";
   #_w39 := #_w38 AND NOT "P_TRIG122";   // rising edge
   "P_TRIG122" := #_w38;
   IF #_w39 THEN "AsansorKapatKat2" := TRUE; END_IF;
   #_w40 := #_w35 AND "Asansor3katta" AND "KapıAcık";
   #_w41 := #_w40 AND NOT "P_TRIG123";   // rising edge
   "P_TRIG123" := #_w40;
   IF #_w41 THEN "AsansorAcKat3" := FALSE; END_IF;
   #_w42 := #_w40 AND "IsıkBariyeri";
   #_w43 := #_w42 AND NOT "P_TRIG124";   // rising edge
   "P_TRIG124" := #_w42;
   IF #_w43 THEN "AsansorKapatKat3" := TRUE; END_IF;
   #_w44 := #_w35 AND "Asansor0katta" AND "KapıAcık";
   #_w45 := #_w44 AND NOT "P_TRIG125";   // rising edge
   "P_TRIG125" := #_w44;
   IF #_w45 THEN "AsansorAcKat0" := FALSE; END_IF;
   #_w46 := #_w44 AND "IsıkBariyeri";
   #_w47 := #_w46 AND NOT "P_TRIG126";   // rising edge
   "P_TRIG126" := #_w46;
   IF #_w47 THEN "AsansorKapatKat0" := TRUE; END_IF;
   #_w48 := 1 AND "AsansorKapatKat2" AND "Asansor2katta" AND "KapıKapalı";
   #_w49 := #_w48 AND NOT "P_TRIG127";   // rising edge
   "P_TRIG127" := #_w48;
   IF #_w49 THEN "AsansorKapatKat2" := FALSE; END_IF;
   #_w50 := 1 AND "AsansorKapatKat3" AND "Asansor3katta" AND "KapıKapalı";
   #_w51 := #_w50 AND NOT "P_TRIG128";   // rising edge
   "P_TRIG128" := #_w50;
   IF #_w51 THEN "AsansorKapatKat3" := FALSE; END_IF;
   #_w52 := 1 AND "AsansorKapatKat0" AND "Asansor0katta" AND "KapıKapalı";
   #_w53 := #_w52 AND NOT "P_TRIG129";   // rising edge
   "P_TRIG129" := #_w52;
   IF #_w53 THEN "AsansorKapatKat0" := FALSE; END_IF;
END_REGION

REGION Network 3
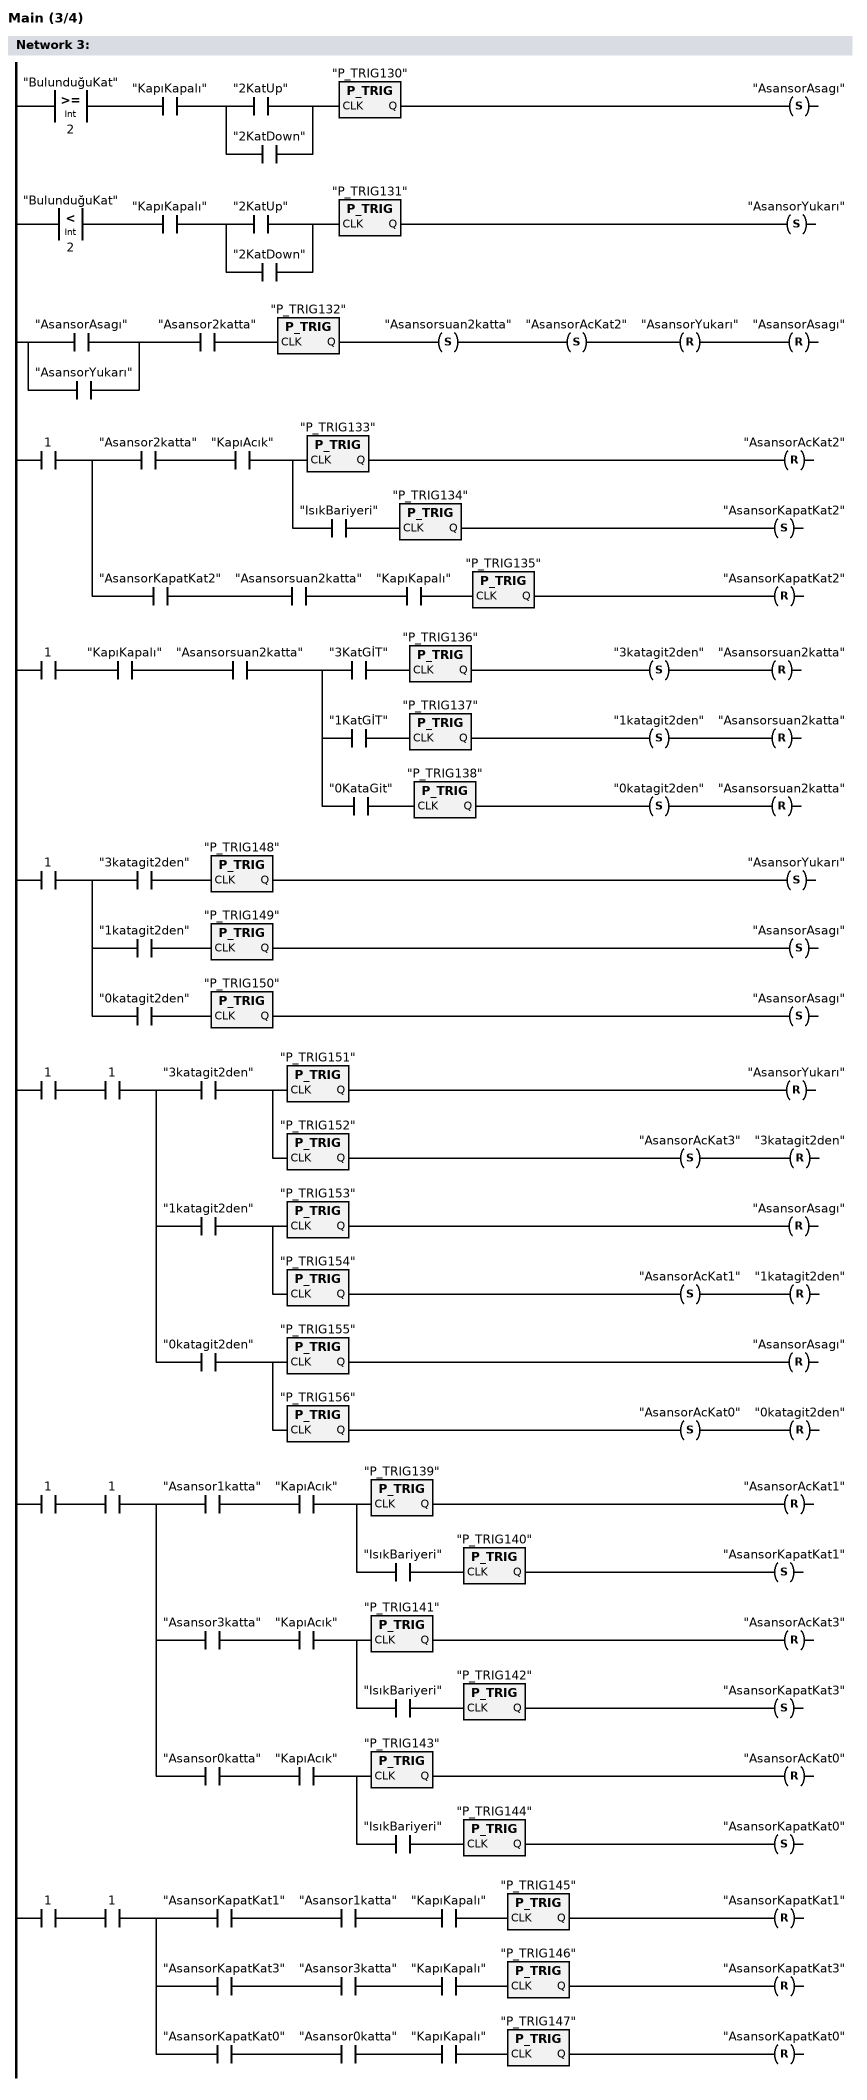
   RUNG wire#powerrail
      { S7_Templates := "SrcType := Int" } GE_Contact(in1 := "BulunduğuKat", in2 := 2)
      Contact( "KapıKapalı" )
      wire#w1
      Contact( "2KatUp" )
      wire#w2
      P_Trig( "P_TRIG130" )
      S_Coil( "AsansorAsagı" )
   END_RUNG
   RUNG wire#w1
      Contact( "2KatDown" )
   END_RUNG wire#w2
   RUNG wire#powerrail
      { S7_Templates := "SrcType := Int" } LT_Contact(in1 := "BulunduğuKat", in2 := 2)
      Contact( "KapıKapalı" )
      wire#w3
      Contact( "2KatUp" )
      wire#w4
      P_Trig( "P_TRIG131" )
      S_Coil( "AsansorYukarı" )
   END_RUNG
   RUNG wire#w3
      Contact( "2KatDown" )
   END_RUNG wire#w4
   RUNG wire#powerrail
      Contact( "AsansorAsagı" )
      wire#w5
      Contact( "Asansor2katta" )
      P_Trig( "P_TRIG132" )
      S_Coil( "Asansorsuan2katta" )
      S_Coil( "AsansorAcKat2" )
      R_Coil( "AsansorYukarı" )
      R_Coil( "AsansorAsagı" )
   END_RUNG
   RUNG wire#powerrail
      Contact( "AsansorYukarı" )
   END_RUNG wire#w5
   RUNG wire#powerrail
      Contact( 1 )
      wire#w6
      Contact( "Asansor2katta" )
      Contact( "KapıAcık" )
      wire#w7
      P_Trig( "P_TRIG133" )
      R_Coil( "AsansorAcKat2" )
   END_RUNG
   RUNG wire#w7
      Contact( "IsıkBariyeri" )
      P_Trig( "P_TRIG134" )
      S_Coil( "AsansorKapatKat2" )
   END_RUNG
   RUNG wire#w6
      Contact( "AsansorKapatKat2" )
      Contact( "Asansorsuan2katta" )
      Contact( "KapıKapalı" )
      P_Trig( "P_TRIG135" )
      R_Coil( "AsansorKapatKat2" )
   END_RUNG
   RUNG wire#powerrail
      Contact( 1 )
      Contact( "KapıKapalı" )
      Contact( "Asansorsuan2katta" )
      wire#w8
      Contact( "3KatGİT" )
      P_Trig( "P_TRIG136" )
      S_Coil( "3katagit2den" )
      R_Coil( "Asansorsuan2katta" )
   END_RUNG
   RUNG wire#w8
      Contact( "1KatGİT" )
      P_Trig( "P_TRIG137" )
      S_Coil( "1katagit2den" )
      R_Coil( "Asansorsuan2katta" )
   END_RUNG
   RUNG wire#w8
      Contact( "0KataGit" )
      P_Trig( "P_TRIG138" )
      S_Coil( "0katagit2den" )
      R_Coil( "Asansorsuan2katta" )
   END_RUNG
   RUNG wire#powerrail
      Contact( 1 )
      wire#w9
      Contact( "3katagit2den" )
      P_Trig( "P_TRIG148" )
      S_Coil( "AsansorYukarı" )
   END_RUNG
   RUNG wire#w9
      Contact( "1katagit2den" )
      P_Trig( "P_TRIG149" )
      S_Coil( "AsansorAsagı" )
   END_RUNG
   RUNG wire#w9
      Contact( "0katagit2den" )
      P_Trig( "P_TRIG150" )
      S_Coil( "AsansorAsagı" )
   END_RUNG
   RUNG wire#powerrail
      Contact( 1 )
      Contact( 1 )
      wire#w10
      Contact( "3katagit2den" )
      wire#w11
      P_Trig( "P_TRIG151" )
      R_Coil( "AsansorYukarı" )
   END_RUNG
   RUNG wire#w11
      P_Trig( "P_TRIG152" )
      S_Coil( "AsansorAcKat3" )
      R_Coil( "3katagit2den" )
   END_RUNG
   RUNG wire#w10
      Contact( "1katagit2den" )
      wire#w12
      P_Trig( "P_TRIG153" )
      R_Coil( "AsansorAsagı" )
   END_RUNG
   RUNG wire#w12
      P_Trig( "P_TRIG154" )
      S_Coil( "AsansorAcKat1" )
      R_Coil( "1katagit2den" )
   END_RUNG
   RUNG wire#w10
      Contact( "0katagit2den" )
      wire#w13
      P_Trig( "P_TRIG155" )
      R_Coil( "AsansorAsagı" )
   END_RUNG
   RUNG wire#w13
      P_Trig( "P_TRIG156" )
      S_Coil( "AsansorAcKat0" )
      R_Coil( "0katagit2den" )
   END_RUNG
   RUNG wire#powerrail
      Contact( 1 )
      Contact( 1 )
      wire#w14
      Contact( "Asansor1katta" )
      Contact( "KapıAcık" )
      wire#w15
      P_Trig( "P_TRIG139" )
      R_Coil( "AsansorAcKat1" )
   END_RUNG
   RUNG wire#w15
      Contact( "IsıkBariyeri" )
      P_Trig( "P_TRIG140" )
      S_Coil( "AsansorKapatKat1" )
   END_RUNG
   RUNG wire#w14
      Contact( "Asansor3katta" )
      Contact( "KapıAcık" )
      wire#w16
      P_Trig( "P_TRIG141" )
      R_Coil( "AsansorAcKat3" )
   END_RUNG
   RUNG wire#w16
      Contact( "IsıkBariyeri" )
      P_Trig( "P_TRIG142" )
      S_Coil( "AsansorKapatKat3" )
   END_RUNG
   RUNG wire#w14
      Contact( "Asansor0katta" )
      Contact( "KapıAcık" )
      wire#w17
      P_Trig( "P_TRIG143" )
      R_Coil( "AsansorAcKat0" )
   END_RUNG
   RUNG wire#w17
      Contact( "IsıkBariyeri" )
      P_Trig( "P_TRIG144" )
      S_Coil( "AsansorKapatKat0" )
   END_RUNG
   RUNG wire#powerrail
      Contact( 1 )
      Contact( 1 )
      wire#w18
      Contact( "AsansorKapatKat1" )
      Contact( "Asansor1katta" )
      Contact( "KapıKapalı" )
      P_Trig( "P_TRIG145" )
      R_Coil( "AsansorKapatKat1" )
   END_RUNG
   RUNG wire#w18
      Contact( "AsansorKapatKat3" )
      Contact( "Asansor3katta" )
      Contact( "KapıKapalı" )
      P_Trig( "P_TRIG146" )
      R_Coil( "AsansorKapatKat3" )
   END_RUNG
   RUNG wire#w18
      Contact( "AsansorKapatKat0" )
      Contact( "Asansor0katta" )
      Contact( "KapıKapalı" )
      P_Trig( "P_TRIG147" )
      R_Coil( "AsansorKapatKat0" )
   END_RUNG
   // the same network as SCL:
   #_w1 := ("BulunduğuKat" >= 2) AND "KapıKapalı" AND ("2KatUp" OR "2KatDown");
   #_w2 := #_w1 AND NOT "P_TRIG130";   // rising edge
   "P_TRIG130" := #_w1;
   IF #_w2 THEN "AsansorAsagı" := TRUE; END_IF;
   #_w3 := ("BulunduğuKat" < 2) AND "KapıKapalı" AND ("2KatUp" OR "2KatDown");
   #_w4 := #_w3 AND NOT "P_TRIG131";   // rising edge
   "P_TRIG131" := #_w3;
   IF #_w4 THEN "AsansorYukarı" := TRUE; END_IF;
   #_w5 := ("AsansorAsagı" OR "AsansorYukarı") AND "Asansor2katta";
   #_w6 := #_w5 AND NOT "P_TRIG132";   // rising edge
   "P_TRIG132" := #_w5;
   IF #_w6 THEN
       "Asansorsuan2katta" := TRUE;
       "AsansorAcKat2" := TRUE;
       "AsansorYukarı" := FALSE;
       "AsansorAsagı" := FALSE;
   END_IF;
   #_w7 := 1 AND "Asansor2katta" AND "KapıAcık";
   #_w8 := #_w7 AND NOT "P_TRIG133";   // rising edge
   "P_TRIG133" := #_w7;
   IF #_w8 THEN "AsansorAcKat2" := FALSE; END_IF;
   #_w9 := #_w7 AND "IsıkBariyeri";
   #_w10 := #_w9 AND NOT "P_TRIG134";   // rising edge
   "P_TRIG134" := #_w9;
   IF #_w10 THEN "AsansorKapatKat2" := TRUE; END_IF;
   #_w11 := 1 AND "AsansorKapatKat2" AND "Asansorsuan2katta" AND "KapıKapalı";
   #_w12 := #_w11 AND NOT "P_TRIG135";   // rising edge
   "P_TRIG135" := #_w11;
   IF #_w12 THEN "AsansorKapatKat2" := FALSE; END_IF;
   #_w13 := 1 AND "KapıKapalı" AND "Asansorsuan2katta";
   #_w14 := #_w13 AND "3KatGİT";
   #_w15 := #_w14 AND NOT "P_TRIG136";   // rising edge
   "P_TRIG136" := #_w14;
   IF #_w15 THEN
       "3katagit2den" := TRUE;
       "Asansorsuan2katta" := FALSE;
   END_IF;
   #_w16 := #_w13 AND "1KatGİT";
   #_w17 := #_w16 AND NOT "P_TRIG137";   // rising edge
   "P_TRIG137" := #_w16;
   IF #_w17 THEN
       "1katagit2den" := TRUE;
       "Asansorsuan2katta" := FALSE;
   END_IF;
   #_w18 := #_w13 AND "0KataGit";
   #_w19 := #_w18 AND NOT "P_TRIG138";   // rising edge
   "P_TRIG138" := #_w18;
   IF #_w19 THEN
       "0katagit2den" := TRUE;
       "Asansorsuan2katta" := FALSE;
   END_IF;
   #_w20 := 1 AND "3katagit2den";
   #_w21 := #_w20 AND NOT "P_TRIG148";   // rising edge
   "P_TRIG148" := #_w20;
   IF #_w21 THEN "AsansorYukarı" := TRUE; END_IF;
   #_w22 := 1 AND "1katagit2den";
   #_w23 := #_w22 AND NOT "P_TRIG149";   // rising edge
   "P_TRIG149" := #_w22;
   IF #_w23 THEN "AsansorAsagı" := TRUE; END_IF;
   #_w24 := 1 AND "0katagit2den";
   #_w25 := #_w24 AND NOT "P_TRIG150";   // rising edge
   "P_TRIG150" := #_w24;
   IF #_w25 THEN "AsansorAsagı" := TRUE; END_IF;
   #_w26 := 1 AND 1;
   #_w27 := #_w26 AND "3katagit2den";
   #_w28 := #_w27 AND NOT "P_TRIG151";   // rising edge
   "P_TRIG151" := #_w27;
   IF #_w28 THEN "AsansorYukarı" := FALSE; END_IF;
   #_w29 := #_w27 AND NOT "P_TRIG152";   // rising edge
   "P_TRIG152" := #_w27;
   IF #_w29 THEN
       "AsansorAcKat3" := TRUE;
       "3katagit2den" := FALSE;
   END_IF;
   #_w30 := #_w26 AND "1katagit2den";
   #_w31 := #_w30 AND NOT "P_TRIG153";   // rising edge
   "P_TRIG153" := #_w30;
   IF #_w31 THEN "AsansorAsagı" := FALSE; END_IF;
   #_w32 := #_w30 AND NOT "P_TRIG154";   // rising edge
   "P_TRIG154" := #_w30;
   IF #_w32 THEN
       "AsansorAcKat1" := TRUE;
       "1katagit2den" := FALSE;
   END_IF;
   #_w33 := #_w26 AND "0katagit2den";
   #_w34 := #_w33 AND NOT "P_TRIG155";   // rising edge
   "P_TRIG155" := #_w33;
   IF #_w34 THEN "AsansorAsagı" := FALSE; END_IF;
   #_w35 := #_w33 AND NOT "P_TRIG156";   // rising edge
   "P_TRIG156" := #_w33;
   IF #_w35 THEN
       "AsansorAcKat0" := TRUE;
       "0katagit2den" := FALSE;
   END_IF;
   #_w36 := 1 AND 1;
   #_w37 := #_w36 AND "Asansor1katta" AND "KapıAcık";
   #_w38 := #_w37 AND NOT "P_TRIG139";   // rising edge
   "P_TRIG139" := #_w37;
   IF #_w38 THEN "AsansorAcKat1" := FALSE; END_IF;
   #_w39 := #_w37 AND "IsıkBariyeri";
   #_w40 := #_w39 AND NOT "P_TRIG140";   // rising edge
   "P_TRIG140" := #_w39;
   IF #_w40 THEN "AsansorKapatKat1" := TRUE; END_IF;
   #_w41 := #_w36 AND "Asansor3katta" AND "KapıAcık";
   #_w42 := #_w41 AND NOT "P_TRIG141";   // rising edge
   "P_TRIG141" := #_w41;
   IF #_w42 THEN "AsansorAcKat3" := FALSE; END_IF;
   #_w43 := #_w41 AND "IsıkBariyeri";
   #_w44 := #_w43 AND NOT "P_TRIG142";   // rising edge
   "P_TRIG142" := #_w43;
   IF #_w44 THEN "AsansorKapatKat3" := TRUE; END_IF;
   #_w45 := #_w36 AND "Asansor0katta" AND "KapıAcık";
   #_w46 := #_w45 AND NOT "P_TRIG143";   // rising edge
   "P_TRIG143" := #_w45;
   IF #_w46 THEN "AsansorAcKat0" := FALSE; END_IF;
   #_w47 := #_w45 AND "IsıkBariyeri";
   #_w48 := #_w47 AND NOT "P_TRIG144";   // rising edge
   "P_TRIG144" := #_w47;
   IF #_w48 THEN "AsansorKapatKat0" := TRUE; END_IF;
   #_w49 := 1 AND 1;
   #_w50 := #_w49 AND "AsansorKapatKat1" AND "Asansor1katta" AND "KapıKapalı";
   #_w51 := #_w50 AND NOT "P_TRIG145";   // rising edge
   "P_TRIG145" := #_w50;
   IF #_w51 THEN "AsansorKapatKat1" := FALSE; END_IF;
   #_w52 := #_w49 AND "AsansorKapatKat3" AND "Asansor3katta" AND "KapıKapalı";
   #_w53 := #_w52 AND NOT "P_TRIG146";   // rising edge
   "P_TRIG146" := #_w52;
   IF #_w53 THEN "AsansorKapatKat3" := FALSE; END_IF;
   #_w54 := #_w49 AND "AsansorKapatKat0" AND "Asansor0katta" AND "KapıKapalı";
   #_w55 := #_w54 AND NOT "P_TRIG147";   // rising edge
   "P_TRIG147" := #_w54;
   IF #_w55 THEN "AsansorKapatKat0" := FALSE; END_IF;
END_REGION

REGION Network 4
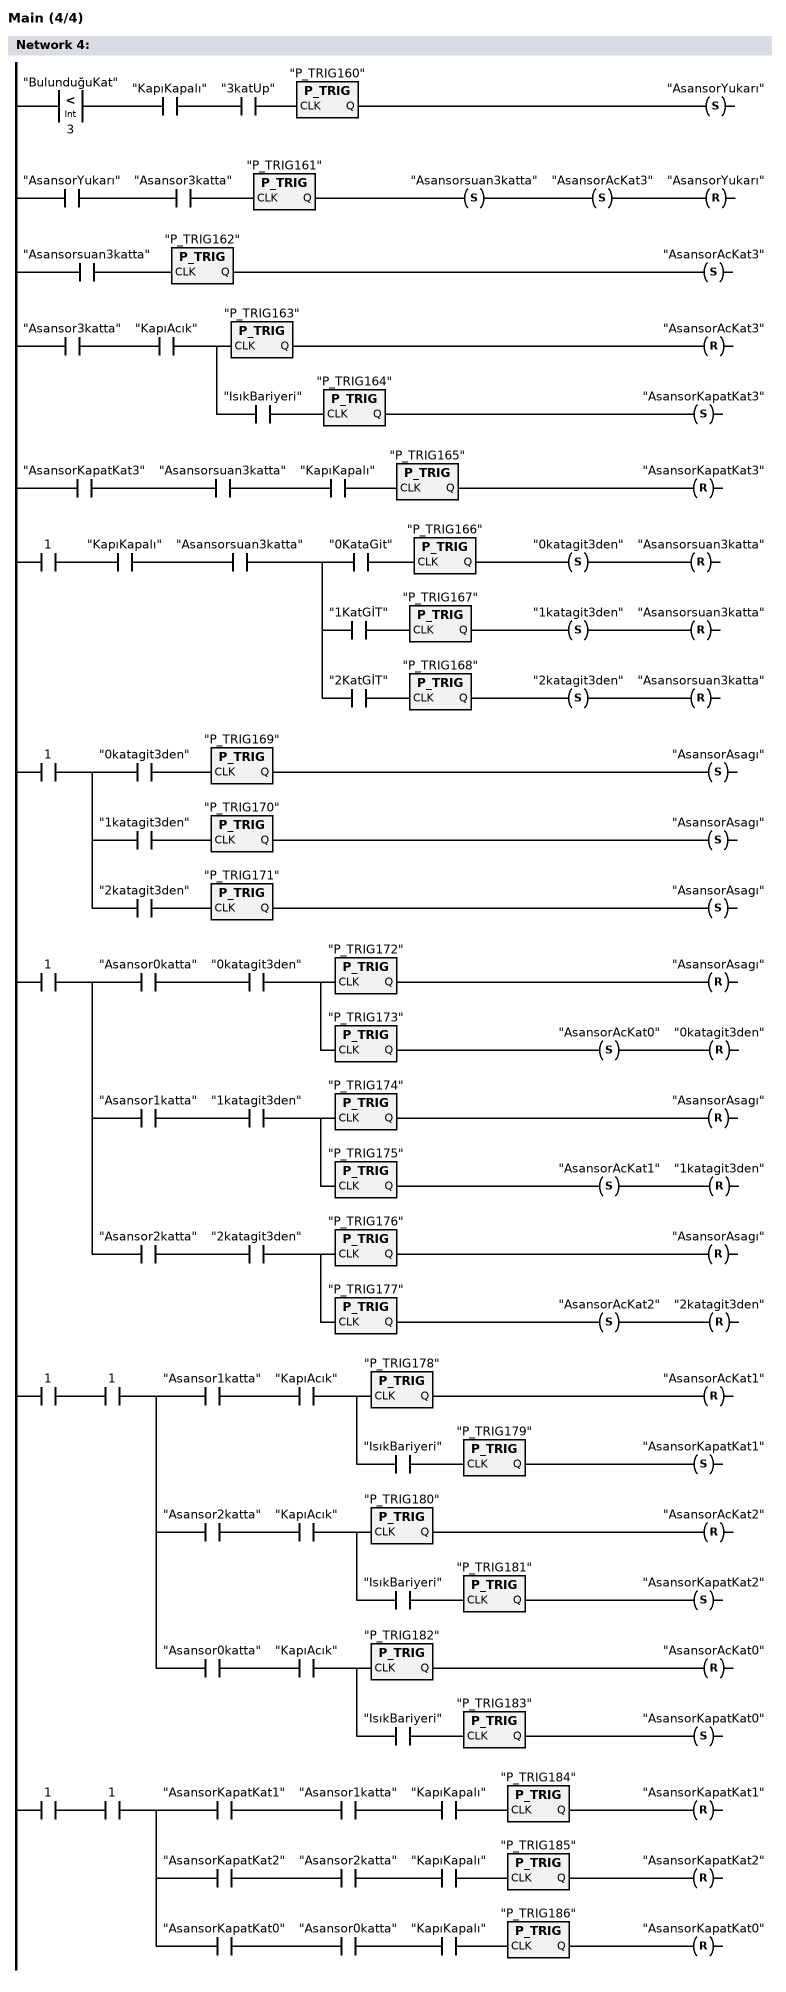
   RUNG wire#powerrail
      { S7_Templates := "SrcType := Int" } LT_Contact(in1 := "BulunduğuKat", in2 := 3)
      Contact( "KapıKapalı" )
      Contact( "3katUp" )
      P_Trig( "P_TRIG160" )
      S_Coil( "AsansorYukarı" )
   END_RUNG
   RUNG wire#powerrail
      Contact( "AsansorYukarı" )
      Contact( "Asansor3katta" )
      P_Trig( "P_TRIG161" )
      S_Coil( "Asansorsuan3katta" )
      S_Coil( "AsansorAcKat3" )
      R_Coil( "AsansorYukarı" )
   END_RUNG
   RUNG wire#powerrail
      Contact( "Asansorsuan3katta" )
      P_Trig( "P_TRIG162" )
      S_Coil( "AsansorAcKat3" )
   END_RUNG
   RUNG wire#powerrail
      Contact( "Asansor3katta" )
      Contact( "KapıAcık" )
      wire#w1
      P_Trig( "P_TRIG163" )
      R_Coil( "AsansorAcKat3" )
   END_RUNG
   RUNG wire#w1
      Contact( "IsıkBariyeri" )
      P_Trig( "P_TRIG164" )
      S_Coil( "AsansorKapatKat3" )
   END_RUNG
   RUNG wire#powerrail
      Contact( "AsansorKapatKat3" )
      Contact( "Asansorsuan3katta" )
      Contact( "KapıKapalı" )
      P_Trig( "P_TRIG165" )
      R_Coil( "AsansorKapatKat3" )
   END_RUNG
   RUNG wire#powerrail
      Contact( 1 )
      Contact( "KapıKapalı" )
      Contact( "Asansorsuan3katta" )
      wire#w2
      Contact( "0KataGit" )
      P_Trig( "P_TRIG166" )
      S_Coil( "0katagit3den" )
      R_Coil( "Asansorsuan3katta" )
   END_RUNG
   RUNG wire#w2
      Contact( "1KatGİT" )
      P_Trig( "P_TRIG167" )
      S_Coil( "1katagit3den" )
      R_Coil( "Asansorsuan3katta" )
   END_RUNG
   RUNG wire#w2
      Contact( "2KatGİT" )
      P_Trig( "P_TRIG168" )
      S_Coil( "2katagit3den" )
      R_Coil( "Asansorsuan3katta" )
   END_RUNG
   RUNG wire#powerrail
      Contact( 1 )
      wire#w3
      Contact( "0katagit3den" )
      P_Trig( "P_TRIG169" )
      S_Coil( "AsansorAsagı" )
   END_RUNG
   RUNG wire#w3
      Contact( "1katagit3den" )
      P_Trig( "P_TRIG170" )
      S_Coil( "AsansorAsagı" )
   END_RUNG
   RUNG wire#w3
      Contact( "2katagit3den" )
      P_Trig( "P_TRIG171" )
      S_Coil( "AsansorAsagı" )
   END_RUNG
   RUNG wire#powerrail
      Contact( 1 )
      wire#w4
      Contact( "Asansor0katta" )
      Contact( "0katagit3den" )
      wire#w5
      P_Trig( "P_TRIG172" )
      R_Coil( "AsansorAsagı" )
   END_RUNG
   RUNG wire#w5
      P_Trig( "P_TRIG173" )
      S_Coil( "AsansorAcKat0" )
      R_Coil( "0katagit3den" )
   END_RUNG
   RUNG wire#w4
      Contact( "Asansor1katta" )
      Contact( "1katagit3den" )
      wire#w6
      P_Trig( "P_TRIG174" )
      R_Coil( "AsansorAsagı" )
   END_RUNG
   RUNG wire#w6
      P_Trig( "P_TRIG175" )
      S_Coil( "AsansorAcKat1" )
      R_Coil( "1katagit3den" )
   END_RUNG
   RUNG wire#w4
      Contact( "Asansor2katta" )
      Contact( "2katagit3den" )
      wire#w7
      P_Trig( "P_TRIG176" )
      R_Coil( "AsansorAsagı" )
   END_RUNG
   RUNG wire#w7
      P_Trig( "P_TRIG177" )
      S_Coil( "AsansorAcKat2" )
      R_Coil( "2katagit3den" )
   END_RUNG
   RUNG wire#powerrail
      Contact( 1 )
      Contact( 1 )
      wire#w8
      Contact( "Asansor1katta" )
      Contact( "KapıAcık" )
      wire#w9
      P_Trig( "P_TRIG178" )
      R_Coil( "AsansorAcKat1" )
   END_RUNG
   RUNG wire#w9
      Contact( "IsıkBariyeri" )
      P_Trig( "P_TRIG179" )
      S_Coil( "AsansorKapatKat1" )
   END_RUNG
   RUNG wire#w8
      Contact( "Asansor2katta" )
      Contact( "KapıAcık" )
      wire#w10
      P_Trig( "P_TRIG180" )
      R_Coil( "AsansorAcKat2" )
   END_RUNG
   RUNG wire#w10
      Contact( "IsıkBariyeri" )
      P_Trig( "P_TRIG181" )
      S_Coil( "AsansorKapatKat2" )
   END_RUNG
   RUNG wire#w8
      Contact( "Asansor0katta" )
      Contact( "KapıAcık" )
      wire#w11
      P_Trig( "P_TRIG182" )
      R_Coil( "AsansorAcKat0" )
   END_RUNG
   RUNG wire#w11
      Contact( "IsıkBariyeri" )
      P_Trig( "P_TRIG183" )
      S_Coil( "AsansorKapatKat0" )
   END_RUNG
   RUNG wire#powerrail
      Contact( 1 )
      Contact( 1 )
      wire#w12
      Contact( "AsansorKapatKat1" )
      Contact( "Asansor1katta" )
      Contact( "KapıKapalı" )
      P_Trig( "P_TRIG184" )
      R_Coil( "AsansorKapatKat1" )
   END_RUNG
   RUNG wire#w12
      Contact( "AsansorKapatKat2" )
      Contact( "Asansor2katta" )
      Contact( "KapıKapalı" )
      P_Trig( "P_TRIG185" )
      R_Coil( "AsansorKapatKat2" )
   END_RUNG
   RUNG wire#w12
      Contact( "AsansorKapatKat0" )
      Contact( "Asansor0katta" )
      Contact( "KapıKapalı" )
      P_Trig( "P_TRIG186" )
      R_Coil( "AsansorKapatKat0" )
   END_RUNG
   // the same network as SCL:
   #_w1 := ("BulunduğuKat" < 3) AND "KapıKapalı" AND "3katUp";
   #_w2 := #_w1 AND NOT "P_TRIG160";   // rising edge
   "P_TRIG160" := #_w1;
   IF #_w2 THEN "AsansorYukarı" := TRUE; END_IF;
   #_w3 := "AsansorYukarı" AND "Asansor3katta";
   #_w4 := #_w3 AND NOT "P_TRIG161";   // rising edge
   "P_TRIG161" := #_w3;
   IF #_w4 THEN
       "Asansorsuan3katta" := TRUE;
       "AsansorAcKat3" := TRUE;
       "AsansorYukarı" := FALSE;
   END_IF;
   #_w5 := "Asansorsuan3katta" AND NOT "P_TRIG162";   // rising edge
   "P_TRIG162" := "Asansorsuan3katta";
   IF #_w5 THEN "AsansorAcKat3" := TRUE; END_IF;
   #_w6 := "Asansor3katta" AND "KapıAcık";
   #_w7 := #_w6 AND NOT "P_TRIG163";   // rising edge
   "P_TRIG163" := #_w6;
   IF #_w7 THEN "AsansorAcKat3" := FALSE; END_IF;
   #_w8 := #_w6 AND "IsıkBariyeri";
   #_w9 := #_w8 AND NOT "P_TRIG164";   // rising edge
   "P_TRIG164" := #_w8;
   IF #_w9 THEN "AsansorKapatKat3" := TRUE; END_IF;
   #_w10 := "AsansorKapatKat3" AND "Asansorsuan3katta" AND "KapıKapalı";
   #_w11 := #_w10 AND NOT "P_TRIG165";   // rising edge
   "P_TRIG165" := #_w10;
   IF #_w11 THEN "AsansorKapatKat3" := FALSE; END_IF;
   #_w12 := 1 AND "KapıKapalı" AND "Asansorsuan3katta";
   #_w13 := #_w12 AND "0KataGit";
   #_w14 := #_w13 AND NOT "P_TRIG166";   // rising edge
   "P_TRIG166" := #_w13;
   IF #_w14 THEN
       "0katagit3den" := TRUE;
       "Asansorsuan3katta" := FALSE;
   END_IF;
   #_w15 := #_w12 AND "1KatGİT";
   #_w16 := #_w15 AND NOT "P_TRIG167";   // rising edge
   "P_TRIG167" := #_w15;
   IF #_w16 THEN
       "1katagit3den" := TRUE;
       "Asansorsuan3katta" := FALSE;
   END_IF;
   #_w17 := #_w12 AND "2KatGİT";
   #_w18 := #_w17 AND NOT "P_TRIG168";   // rising edge
   "P_TRIG168" := #_w17;
   IF #_w18 THEN
       "2katagit3den" := TRUE;
       "Asansorsuan3katta" := FALSE;
   END_IF;
   #_w19 := 1 AND "0katagit3den";
   #_w20 := #_w19 AND NOT "P_TRIG169";   // rising edge
   "P_TRIG169" := #_w19;
   IF #_w20 THEN "AsansorAsagı" := TRUE; END_IF;
   #_w21 := 1 AND "1katagit3den";
   #_w22 := #_w21 AND NOT "P_TRIG170";   // rising edge
   "P_TRIG170" := #_w21;
   IF #_w22 THEN "AsansorAsagı" := TRUE; END_IF;
   #_w23 := 1 AND "2katagit3den";
   #_w24 := #_w23 AND NOT "P_TRIG171";   // rising edge
   "P_TRIG171" := #_w23;
   IF #_w24 THEN "AsansorAsagı" := TRUE; END_IF;
   #_w25 := 1 AND "Asansor0katta" AND "0katagit3den";
   #_w26 := #_w25 AND NOT "P_TRIG172";   // rising edge
   "P_TRIG172" := #_w25;
   IF #_w26 THEN "AsansorAsagı" := FALSE; END_IF;
   #_w27 := #_w25 AND NOT "P_TRIG173";   // rising edge
   "P_TRIG173" := #_w25;
   IF #_w27 THEN
       "AsansorAcKat0" := TRUE;
       "0katagit3den" := FALSE;
   END_IF;
   #_w28 := 1 AND "Asansor1katta" AND "1katagit3den";
   #_w29 := #_w28 AND NOT "P_TRIG174";   // rising edge
   "P_TRIG174" := #_w28;
   IF #_w29 THEN "AsansorAsagı" := FALSE; END_IF;
   #_w30 := #_w28 AND NOT "P_TRIG175";   // rising edge
   "P_TRIG175" := #_w28;
   IF #_w30 THEN
       "AsansorAcKat1" := TRUE;
       "1katagit3den" := FALSE;
   END_IF;
   #_w31 := 1 AND "Asansor2katta" AND "2katagit3den";
   #_w32 := #_w31 AND NOT "P_TRIG176";   // rising edge
   "P_TRIG176" := #_w31;
   IF #_w32 THEN "AsansorAsagı" := FALSE; END_IF;
   #_w33 := #_w31 AND NOT "P_TRIG177";   // rising edge
   "P_TRIG177" := #_w31;
   IF #_w33 THEN
       "AsansorAcKat2" := TRUE;
       "2katagit3den" := FALSE;
   END_IF;
   #_w34 := 1 AND 1;
   #_w35 := #_w34 AND "Asansor1katta" AND "KapıAcık";
   #_w36 := #_w35 AND NOT "P_TRIG178";   // rising edge
   "P_TRIG178" := #_w35;
   IF #_w36 THEN "AsansorAcKat1" := FALSE; END_IF;
   #_w37 := #_w35 AND "IsıkBariyeri";
   #_w38 := #_w37 AND NOT "P_TRIG179";   // rising edge
   "P_TRIG179" := #_w37;
   IF #_w38 THEN "AsansorKapatKat1" := TRUE; END_IF;
   #_w39 := #_w34 AND "Asansor2katta" AND "KapıAcık";
   #_w40 := #_w39 AND NOT "P_TRIG180";   // rising edge
   "P_TRIG180" := #_w39;
   IF #_w40 THEN "AsansorAcKat2" := FALSE; END_IF;
   #_w41 := #_w39 AND "IsıkBariyeri";
   #_w42 := #_w41 AND NOT "P_TRIG181";   // rising edge
   "P_TRIG181" := #_w41;
   IF #_w42 THEN "AsansorKapatKat2" := TRUE; END_IF;
   #_w43 := #_w34 AND "Asansor0katta" AND "KapıAcık";
   #_w44 := #_w43 AND NOT "P_TRIG182";   // rising edge
   "P_TRIG182" := #_w43;
   IF #_w44 THEN "AsansorAcKat0" := FALSE; END_IF;
   #_w45 := #_w43 AND "IsıkBariyeri";
   #_w46 := #_w45 AND NOT "P_TRIG183";   // rising edge
   "P_TRIG183" := #_w45;
   IF #_w46 THEN "AsansorKapatKat0" := TRUE; END_IF;
   #_w47 := 1 AND 1;
   #_w48 := #_w47 AND "AsansorKapatKat1" AND "Asansor1katta" AND "KapıKapalı";
   #_w49 := #_w48 AND NOT "P_TRIG184";   // rising edge
   "P_TRIG184" := #_w48;
   IF #_w49 THEN "AsansorKapatKat1" := FALSE; END_IF;
   #_w50 := #_w47 AND "AsansorKapatKat2" AND "Asansor2katta" AND "KapıKapalı";
   #_w51 := #_w50 AND NOT "P_TRIG185";   // rising edge
   "P_TRIG185" := #_w50;
   IF #_w51 THEN "AsansorKapatKat2" := FALSE; END_IF;
   #_w52 := #_w47 AND "AsansorKapatKat0" AND "Asansor0katta" AND "KapıKapalı";
   #_w53 := #_w52 AND NOT "P_TRIG186";   // rising edge
   "P_TRIG186" := #_w52;
   IF #_w53 THEN "AsansorKapatKat0" := FALSE; END_IF;
END_REGION
END_ORGANIZATION_BLOCK

(* ===== HMI "HMI_RT_1" =====
system functions are stored by id; their names below are inferred from use
connection "HMI_Connection_1": ETHERNET, S7_1500_OMS

HMI tags "Default tag table"
   "Tag_ScreenNumber" : UInt, internal
   "Asansor0katta" : Bool = PLC Asansor0katta AT %M2.0, 1 s
   "Asansor1katta" : Bool = PLC Asansor1katta AT %M2.1, 1 s
   "Asansor2katta" : Bool = PLC Asansor2katta AT %M2.3, 1 s
   "Asansor3katta" : Bool = PLC Asansor3katta AT %M2.2, 1 s
   "BulunduğuKat" : Int = PLC BulunduğuKat AT %MW0, 1 s
   "AsansorAsagı" : Bool = PLC AsansorAsagı AT %M2.5, 1 s
   "KapıAcık" : Bool = PLC KapıAcık AT %M3.0, 1 s
   "KapıKapalı" : Bool = PLC KapıKapalı AT %M3.4, 1 s
   "AsansorAcKat0" : Bool = PLC AsansorAcKat0 AT %M2.7, 1 s
   "AsansorKapatKat0" : Bool = PLC AsansorKapatKat0 AT %M3.2, 1 s
   "IsıkBariyeri" : Bool = PLC IsıkBariyeri AT %M3.5, 1 s
   "0KatDown" : Bool = PLC 0KatDown AT %M3.6, 1 s
   "1KatGİT" : Bool = PLC 1KatGİT AT %M4.0, 1 s
   "2KatGİT" : Bool = PLC 2KatGİT AT %M4.1, 1 s
   "3KatGİT" : Bool = PLC 3KatGİT AT %M4.2, 1 s
   "AsansorAcKat1" : Bool = PLC AsansorAcKat1 AT %M4.5, 1 s
   "AsansorKapatKat1" : Bool = PLC AsansorKapatKat1 AT %M4.7, 1 s
   "AsansorYukarı" : Bool = PLC AsansorYukarı AT %M4.3, 1 s
   "AsansorAcKat2" : Bool = PLC AsansorAcKat2 AT %M5.3, 1 s
   "AsansorKapatKat2" : Bool = PLC AsansorKapatKat2 AT %M6.7, 1 s
   "AsansorAcKat3" : Bool = PLC AsansorAcKat3 AT %M5.6, 1 s
   "AsansorKapatKat3" : Bool = PLC AsansorKapatKat3 AT %M7.0, 1 s
   "1KatUp" : Bool = PLC 1KatUp AT %M7.7, 1 s
   "1KatDown" : Bool = PLC 1KatDown AT %M7.5, 1 s
   "0KataGit" : Bool = PLC 0KataGit AT %M8.4, 1 s
   "2KatUp" : Bool = PLC 2KatUp AT %M25.0, 1 s
   "2KatDown" : Bool = PLC 2KatDown AT %M24.7, 1 s
   "3katUp" : Bool = PLC 3katUp AT %M20.7, 1 s

screen "Root screen" 1280x740, template "Template_1"
   on GenerateScreen: SetTag("Tag_ScreenNumber", 1)
   Button "Button_1" at 8,29 size 218x32; TextOff 'Asansor 0. Katta Sensör'
      on Press: InvertBit("Asansor0katta")
   Button "Button_2" at 4,76 size 218x32; TextOff 'Asansor 1. Katta Sensör'
      on Press: InvertBit("Asansor1katta")
   Button "Button_3" at 8,126 size 218x32; TextOff 'Asansor 2. Katta Sensör'
      on Press: InvertBit("Asansor2katta")
   Button "Button_4" at 8,171 size 218x32; TextOff 'Asansor 3. Katta Sensör'
      on Press: InvertBit("Asansor3katta")
   Ellipse "Ellipse_1" at 233,21 size 96x41
      Appearance <- "Asansor0katta"
   Ellipse "Ellipse_2" at 233,61 size 96x41
      Appearance <- "Asansor1katta"
   Ellipse "Ellipse_3" at 240,113 size 96x41
      Appearance <- "Asansor2katta"
   Ellipse "Ellipse_4" at 241,163 size 96x41
      Appearance <- "Asansor3katta"
   TextField "Text field_1" at 475,21 size 236x25; Text 'Bulunduğu Kat Bilgisi: 0'
   TextField "Text field_2" at 475,75 size 236x25; Text 'Bulunduğu Kat Bilgisi: 1'
   TextField "Text field_3" at 475,129 size 236x25; Text 'Bulunduğu Kat Bilgisi: 2'
   TextField "Text field_4" at 475,183 size 236x25; Text 'Bulunduğu Kat Bilgisi: 3'
   Ellipse "Ellipse_5" at 701,14 size 96x48
      Appearance <- "BulunduğuKat"
   Ellipse "Ellipse_6" at 701,65 size 96x48
      Appearance <- "BulunduğuKat"
   Ellipse "Ellipse_7" at 700,113 size 96x48
      Appearance <- "BulunduğuKat"
   Ellipse "Ellipse_8" at 701,160 size 96x48
      Appearance <- "BulunduğuKat"
   TextField "Text field_5" at 8,228 size 152x25; Text 'Asansor Asagı :'
   TextField "Text field_6" at 0,277 size 160x25; Text 'Asansor Yukarı :'
   Ellipse "Ellipse_9" at 160,214 size 96x48
      Appearance <- "AsansorAsagı"
   Ellipse "Ellipse_10" at 160,267 size 96x48
      Appearance <- "AsansorYukarı"
   Ellipse "Ellipse_11" at 121,315 size 96x48
      Appearance <- "KapıAcık"
   Ellipse "Ellipse_12" at 123,370 size 96x48
      Appearance <- "KapıKapalı"
   Button "Button_5" at 4,318 size 96x32; TextOff 'Kapı Acık:'
      on Press: InvertBit("KapıAcık")
   Button "Button_6" at 8,378 size 96x32; TextOff 'Kapı Kapalı:'
      on Press: InvertBit("KapıKapalı")
   TextField "Text field_7" at 475,235 size 173x25; Text 'Asansor Ac Kat 0:'
   TextField "Text field_8" at 479,271 size 205x25; Text 'Asansor Kapat Kat 0:'
   Ellipse "Ellipse_13" at 654,212 size 96x48
      Appearance <- "AsansorAcKat0"
   Ellipse "Ellipse_14" at 675,260 size 96x48
      Appearance <- "AsansorKapatKat0"
   TextField "Text field_9" at 12,451 size 17x25; Text 'Text'
   Button "Button_7" at 8,451 size 127x32; TextOff 'IsıkBariyeri'
      on Press: InvertBit("IsıkBariyeri")
   Ellipse "Ellipse_15" at 150,442 size 96x48
      Appearance <- "IsıkBariyeri"
   Button "Button_8" at 12,518 size 159x32; TextOff '0.Kat Down'
      Appearance <- "0KatDown"
      on Press: function_b14e0dd5("0KatDown", 0)
   GraphicIOField "Graphic I/O field_1" at 805,165 size 341x401
   Button "Button_9" at 838,318 size 96x32; TextOff '3.Kat'
      on Press: function_b14e0dd5("3KatGİT", 0)
   Button "Button_10" at 841,372 size 96x32; TextOff '2.Kat'
      on Press: function_b14e0dd5("2KatGİT", 0)
   Button "Button_11" at 839,429 size 96x32; TextOff '1Kat'
      on Press: function_b14e0dd5("1KatGİT", 0)
   TextField "Text field_10" at 477,331 size 173x25; Text 'Asansor Ac Kat 1:'
   TextField "Text field_11" at 481,367 size 205x25; Text 'Asansor Kapat Kat 1:'
   Ellipse "Ellipse_16" at 656,308 size 96x48
      Appearance <- "AsansorAcKat1"
   Ellipse "Ellipse_17" at 677,356 size 96x48
      Appearance <- "AsansorKapatKat1"
   TextField "Text field_12" at 477,436 size 173x25; Text 'Asansor Ac Kat 2:'
   TextField "Text field_13" at 481,472 size 205x25; Text 'Asansor Kapat Kat 2:'
   Ellipse "Ellipse_18" at 656,413 size 96x48
      Appearance <- "AsansorAcKat2"
   Ellipse "Ellipse_19" at 677,461 size 96x48
      Appearance <- "AsansorKapatKat2"
   TextField "Text field_14" at 477,541 size 173x25; Text 'Asansor Ac Kat 3:'
   TextField "Text field_15" at 481,577 size 205x25; Text 'Asansor Kapat Kat 3:'
   Ellipse "Ellipse_20" at 656,518 size 96x48
      Appearance <- "AsansorAcKat3"
   Ellipse "Ellipse_21" at 677,566 size 96x48
      Appearance <- "AsansorKapatKat3"
   Button "Button_14" at 839,497 size 96x32; TextOff '0.kat'
      on Press: function_b14e0dd5("0KataGit", 0)
   Button "Button_12" at 14,563 size 96x32; TextOff '1.Kat Up'
      on Press: function_b14e0dd5("1KatUp", 0)
   Button "Button_13" at 123,563 size 100x32; TextOff '1.Kat Down'
      on Press: function_b14e0dd5("1KatDown", 0)
   Button "Button_15" at 8,602 size 96x32; TextOff '2.Kat Up'
      on Press: function_b14e0dd5("2KatUp", 0)
   Button "Button_16" at 123,606 size 96x32; TextOff '2.Kat Down'
      on Press: function_b14e0dd5("2KatDown", 0)
   Button "Button_17" at 12,647 size 96x32; TextOff '3.KatUp'
      on Press: function_b14e0dd5("3katUp", 0)
   Ellipse "Ellipse_22" at 808,203 size 71x48
      Appearance <- "BulunduğuKat"
   Ellipse "Ellipse_23" at 884,203 size 74x48
      Appearance <- "BulunduğuKat"
   Ellipse "Ellipse_24" at 967,202 size 67x48
      Appearance <- "BulunduğuKat"
   Ellipse "Ellipse_25" at 1052,200 size 65x48
      Appearance <- "BulunduğuKat"
   TextField "Text field_16" at 824,169 size 17x25; Text '0'
   TextField "Text field_17" at 913,171 size 17x25; Text '1'
   TextField "Text field_18" at 984,171 size 17x25; Text '2'
   TextField "Text field_19" at 1076,169 size 17x25; Text '3'

Template "Template_1" 1280x740
   Button "Exit" at 1200,679 size 78x59; TextOff 'Exit'; PictureOff "ExitRuntime_TP1200_Comfort_TR"; PictureOn "ExitRuntime_TP1200_Comfort_TR"
      on Release: StopRuntime(0)
   Button "Template_Button" at 1120,679 size 78x59; TextOff 'Text'
   Button "Template_Button_1" at 1040,679 size 78x59; TextOff 'Text'
   Button "Template_Button_2" at 960,679 size 78x59; TextOff 'Text'
   Button "Template_Button_3" at 880,679 size 78x59; TextOff 'Text'
   Button "Template_Button_4" at 800,679 size 78x59; TextOff 'Text'
   Button "Template_Button_5" at 720,679 size 78x59; TextOff 'Text'
   Button "Template_Button_6" at 640,679 size 78x59; TextOff 'Text'
   Button "Template_Button_7" at 561,679 size 78x59; TextOff 'Text'
   Button "Template_Button_8" at 481,679 size 78x59; TextOff 'Text'
   Button "Template_Button_9" at 401,679 size 78x59; TextOff 'Text'
   Button "Template_Button_10" at 321,679 size 78x59; TextOff 'Text'
   Button "Template_Button_11" at 241,679 size 78x59; TextOff 'Text'
   Button "Template_Button_12" at 161,679 size 78x59; TextOff 'Text'
   Button "Alarms" at 81,679 size 78x59; TextOff 'Alarms'; PictureOff "AlarmDisplay_TP1200_Comfort_TR"; PictureOn "AlarmDisplay_TP1200_Comfort_TR"
      on Release: function_ef3f5d25("Alarm window_Unacknowledged", -1)
   Button "Start screen" at 1,679 size 78x59; TextOff 'Start screen'; PictureOff "NavigateHome_TP1200_Comfort_TR"; PictureOn "NavigateHome_TP1200_Comfort_TR"
      on Release: ActivateScreen("Root screen", 0)
*)